IF bAConeOnMatrixConv AND bAutoModeOn AND bErrorReset AND NOT bIRowConeDetection  THEN
sMatrixConvStatus:='Continue Machine Operation '; bAConeOnMatrixConv:=FALSE;END_IF



(*===================== Auto Logic================*)


CASE step4 OF

	0:	IF( bARowStopperMotorRevStart ) AND bAutoModeOn THEN
		bAMove2_4Position:=FALSE;
		bAMove2_3Position:=FALSE;
		bRowStopperAt23Pos:=FALSE;
		bRowStopperAt24Pos:=FALSE;
		tRowStopperHomeDly(IN:=TRUE , PT:= t#1s , Q=> , ET=> );
		IF tRowStopperHomeDly.Q THEN   step4:=step4+1; END_IF
		END_IF

	1:	step4:=step4+1;


	2:	IF tRowStopperHomeDly.Q AND bAutoModeOn  AND NOT bAPauseSeq   THEN
		bQARowStopperMotorRevAuto:=TRUE;
		bARowStopperMotorRevStart:=FALSE;
		TON_2(IN:=FALSE);
		step4:=step4+1;
		END_IF

	3:	 step4:=step4+1;

	4:	IF bAutoModeOn AND bIRowStopperHome  THEN
		bQARowStopperMotorRevAuto:=FALSE;
		bAServoFwdStart:=TRUE;
		bAServoStartAuto:=TRUE;
		tRowStopperHomeDly(IN:=FALSE);
		step4:=step4+1;
		END_IF

	5:	 step4:=step4+1;

	6:	IF  bIGripperVerticalEnd THEN
		step4:=step4+1;
		END_IF

	7:	IF NOT bIGripperVerticalEnd   AND NOT bAPauseSeq   THEN
		step4:=step4+1;
		END_IF


	8:	 step4:=step4+1;

	9:	TON_2(IN:=TRUE , PT:=T#3S , Q=> , ET=> );
		IF TON_2.Q  THEN bAServoUpDone:=TRUE; step4:=step4+1; END_IF

	10:	 step4:=step4+1;


	11:	IF  bAutoModeOn AND  bAServoUpDone  AND b2_4SetHmiSelected THEN
		step4:=12;
		ELSIF  bAutoModeOn AND  bAServoUpDone AND b2_3SetHmiSelected THEN
		step4:=14;
		END_IF


	12:	 step4:=step4+1;

	13:	 bAMove2_4Position:=TRUE;
		step4:=16;

	14:	 step4:=step4+1;

	15:	bAMove2_3Position:=TRUE;
		step4:=step4+1;

	16:	 step4:=step4+1;

	17:	bAServoUpDone:=FALSE;
		step4:=0;

END_CASE

(*

R_TRIG_1(CLK:=b2_3SetHmiSelected , Q=> );


IF R_TRIG_1.Q AND NOT bIRowStopper2 THEN
b2_3FirstMoveStart:=TRUE;

END_IF

*)
(*
R_TRIG_2(CLK:=b2_4SetHmiSelected , Q=> );


IF R_TRIG_2.Q AND NOT bIRowStopper3 THEN
b2_4FirstMoveStart:=TRUE;

END_IF*)



(*============= Row Stopper Go to Home Logic While Servo Reset==========================*)


CASE Step5 OF
	0:	IF bRowStopperGoHome THEN bRowStopperGoRst:=TRUE; step5:=1; END_IF

	1:	IF bIRowStopperHome THEN  bRowStopperGoHome:=FALSE; bRowStopperGoRst:=FALSE; Step5:=0; END_IF

END_CASE


IF NOT bIEmergencySwitch OR bStopHmi   OR bServoOff OR bIMcStop  THEN
TON1temp4(IN:=FALSE);
RevStartT(IN:=FALSE);
bA2_4MoveEnable:=FALSE;
bA2_4RowMoveStarted:=FALSE;
bRowStopperAt24Pos:=FALSE;
bA2_3MoveEnable:=FALSE;
b23CheckDly(IN:=FALSE);
bA2_3MoveStarted:=FALSE;
TON_Mx(IN:=FALSE);
bRowStopperAt23Pos:=FALSE;
bRowStopperIntOver:=FALSE;
bAConeOnMatrixConv1:=FALSE;
bAConeOnMatrixConv2:=FALSE;
bAConeOnMatrixConv:=FALSE;
tRowStopperHomeDly(IN:=FALSE);
TON_2(IN:=FALSE);
bAServoFwdStart:=FALSE;
bAServoUpDone:=FALSE;
bAMove2_4Position:=FALSE;
bAMove2_3Position:=FALSE;

bQARowStopperMotorFwd1:=FALSE;
bQARowStopperMotorFwd2:=FALSE;
bQARowStopperMotorFwd3:=FALSE;
bQARowStopperMotorRev1:=FALSE;
bQARowStopperMotorRev2:=FALSE;
bQARowStopperMotorRev3:=FALSE;
bQARowStopperMotorRevAuto:=FALSE;
bRowStopperGoRst:=FALSE;
step2:=0;
step1:=0;
step3:=0;
step4:=0;

END_IF
END_PROGRAM

(* POU Auto/ColumStopperMotor, ST *)
PROGRAM ColumStopperMotor
VAR
	bQAColumnStopperMotorFwd1: BOOL;
	bQAColumnStopperMotorRev1: BOOL;
	step1: INT;

	test: BOOL;

	step2: INT;
	ColumnStopperInHome: BOOL;
	bA4_4MoveStarted: BOOL;
	bQAColumnStopperMotorFw21: BOOL;
	bQAColumnStopperMotorFwd2: BOOL;
	bQAColumnStopperMotorRev2: BOOL;
	bQAColumnStopperMotorFw2: BOOL;
	test1: BOOL;
	step3: INT;
	test2: BOOL;
	bA2_3MoveStarted: BOOL;
	bQAColumnStopperMotorRev3: BOOL;
	bQAColumnStopperMotorFwd3: BOOL;
	RevOffDly: TON;
	bA2_4MoveStarted: BOOL;
	Timer1: TON;
	Timer2: TON;
	bStopHmitemp: BOOL;
	bProgramChange: BOOL;
	bColumnStopMove2_3: BOOL;
	bColumnStopMove2_4: BOOL;
	b2_3SetHmiSelectedtemp: BOOL;
	b2_4SetHmiSelectedtemp: BOOL;
	b2_4SetHmiSelectedtemp1: BOOL;
	Mybit1: BOOL;
END_VAR
bQAColumnStopperMotorForward:= ( bQAColumnStopperMotorFwd1 OR bQAColumnStopperMotorFwd2 OR bQAColumnStopperMotorFwd3  ) ;
bQAColumnStopperMotorReverse:= ( bQAColumnStopperMotorRev1 ) ;

								(*=========== Column Stopper Motor Home Position Logic===============*)

CASE step2 OF

	0:	IF  bInitializeHmi AND bMCStartInAuto  AND NOT bIColumnStopperHome  AND NOT bAinterlockinit   THEN
		bQAColumnStopperMotorFwd1:=TRUE;
		(*	Timer1(IN:=TRUE  , PT:=t#1s , Q=> , ET=> );   *) step2:=step2+1;
		ELSIF  bInitializeHmi AND  bIColumnStopperHome    THEN   step2:=4;
		END_IF

	1:	bQAColumnStopperMotorFwd1:=FALSE;
		Timer2(IN:=TRUE , PT:= t#0.5s, Q=> , ET=> );
		IF Timer2.Q THEN step2 :=step2+1; END_IF

	2:	IF NOT bAPauseSeq  THEN  bQAColumnStopperMotorRev1:=TRUE; step2:=step2+1; END_IF

	3:	IF bIColumnStopperHome THEN bQAColumnStopperMotorRev1:=FALSE; step2:=step2+1; END_IF

	4:	IF b2_3SetHmiSelected THEN bColumnStopMove2_3:=TRUE; step2:=0;
		ELSIF b2_4SetHmiSelected THEN bColumnStopMove2_4:=TRUE; step2:=0;
		END_IF

END_CASE

										(*=========== Column Stopper Motor 2_3 Position Logic===============*)

CASE step1 OF

	0:	IF  b2_3SetHmiSelected AND bColumnStopMove2_3 AND NOT bIColumnStopper3  AND  bIColumnStopperHome  THEN
		 bQAColumnStopperMotorFwd2:=TRUE; step1:=step1+1;
		END_IF

	1:	IF bIColumnStopper3 THEN
	         bColumnStopMove2_3:=FALSE;
                  bQAColumnStopperMotorFwd2:=FALSE; step1:=step1+1;
		END_IF

	2:	 step1:=0;

END_CASE

										(*=========== Column Stopper Motor 2_4 Position Logic===============*)

CASE step3 OF

	0:	IF b2_4SetHmiSelected AND  bColumnStopMove2_4 AND NOT bIColumnStopper2  AND    bIColumnStopperHome   THEN
		bQAColumnStopperMotorFwd3:=TRUE; step3:=step3+1;
		END_IF


	1: 	IF bIColumnStopper2 THEN
		bColumnStopMove2_4:=FALSE;
		bQAColumnStopperMotorFwd3:=FALSE; step3:=step3+1;
		END_IF


	2:	step3:=0;

END_CASE
END_PROGRAM

(* POU StartUp/GripperUnitRst, ST *)
PROGRAM GripperUnitRst
VAR
	step: INT;
	bILengthTightPistonEnd: BOOL;
	bIBredthTightPistonEnd: BOOL;
	bEmptyCortonConveyoPiatonHome: BOOL;
	bHorPistonAtReadyPos: BOOL;
	bHorPistonAtHomePos: BOOL;
	bHorPistonAtMiddlePos: BOOL;
	bGripperAtHomePos: BOOL;
	bGripperAtEndPos: BOOL;
	bGripperAtMiddlePos: BOOL;
	bSepVerticalAtHomePos: BOOL;
	bSepVerticalAtEndPos: BOOL;
	bSepVerticalAtMiddlePos: BOOL;
	bLenghtTightPistonHomeNok: BOOL;
	bBreathtightPistonHomeNok: BOOL;
	bApplicatorHomeNok: BOOL;
	bReleaseApplicator: BOOL;
	step2: INT;
	Timer1: TON;
	Timer2: TON;
	Timer3: TON;
	Timer4: TON;
	ReadyToRelease: BOOL;
	Timer5: TON;
	bAResetHmitemp: BOOL;
	Timer6: TON;
	Timer7: TON;
	Timer8: TON;
	Timer9: TON;
	test: BOOL;
	BTEST1: BOOL;
	Timer10: TON;
	Timer20: TON;
	check1: BOOL;
	R_TRIG_50: R_TRIG;
END_VAR
VAR_INPUT
END_VAR
IF bInitializeHmi AND bAutoModeOn AND bMCStartInAuto THEN
step:=0;
END_IF



CASE step OF
	0:	 bHomingDone:=FALSE;
		step:=step+1;

	1:	step:=step+1;


	2:	IF  bAResetHmitemp OR bMatrixConvIntOver THEN step:=step+1;  END_IF

	3:	IF NOT bIGripperVerticalHome AND bIServoReady THEN
		bServoStopHmi:=FALSE;
		bServoPwrOff:=FALSE;
		  bRServoHome:=TRUE; step:=step+1;
		ELSIF bIGripperVerticalHome AND bIServoReady  THEN
		step:=step+3;
		END_IF

	4:	IF bHomingDone THEN
		bMatrixConvIntOver:=FALSE;
		 step:=step+1; END_IF

	5:	IF bQALengthTightPistonValve AND bQABreadthTightPistonValve THEN
		bHomingDone:=FALSE;
		step:=step+1;
		ELSIF bQALengthTightPistonValve AND NOT bQABreadthTightPistonValve THEN
		bQABreadthTightPistonValve:=FALSE;
		bQALengthTightPistonValve:=FALSE;
		bQMBreadthTightPistonValve:=FALSE;
		bQMLengthTightPistonValve:=FALSE;

		bHomingDone:=FALSE;

		END_IF
		IF bILengthTightPistonHome THEN
		bQAConeEjectionPistonValve:=FALSE;
		bQMConeEjectionPistonValve:=FALSE;
		IF bIConeEjectionPistonHome THEN
		step:=step+1;
		END_IF
		END_IF
	6:	bMatrixConvIntOver:=FALSE;
		IF bISeparatorHorizontalPistonEnd AND NOT  bISeparatorHorizontalPistonHome THEN
		bHorPistonAtReadyPos:=TRUE; bHorPistonAtHomePos:=FALSE; bHorPistonAtMiddlePos:=FALSE;
		step:=step+1;
		ELSIF NOT bISeparatorHorizontalPistonEnd  AND  bISeparatorHorizontalPistonHome THEN
		bHorPistonAtHomePos:=TRUE; bHorPistonAtReadyPos:=FALSE; bHorPistonAtMiddlePos:=FALSE;
		step:=step+1;
		ELSIF NOT bISeparatorHorizontalPistonEnd  AND  NOT bISeparatorHorizontalPistonHome THEN
		bHorPistonAtMiddlePos:=TRUE; bHorPistonAtHomePos:=FALSE; bHorPistonAtReadyPos:=FALSE;
		step:=step+1;
		END_IF

	7:	IF bHorPistonAtReadyPos THEN step:=8;
		ELSIF bHorPistonAtHomePos THEN step:=25;
		ELSIF bHorPistonAtMiddlePos THEN  step:=25; END_IF

	8:	(* iControlWord1:=0;*)
		step:=step+1;

	9:	(* iControlWord1:=6;*)
		step:=Step+1;
(*========Waiting for row stopper to home==========*)

	10:	IF bIRowStopperHome THEN step:=Step+1;
		ELSIF NOT bIRowStopperHome THEN bRowStopperGoHome:=TRUE;  step:=Step+1;  END_IF


	11:	IF  bIRowStopperHome THEN
		bHomingDone:=FALSE;
		bARampDisableAuto:=FALSE;
		bARampDisableAuto2:=FALSE;
		bARampDisableAuto3:=FALSE;
		bARampDisableAuto4:=FALSE;
		bARampDisableRst:= FALSE;
		bAGoCounterAuto:=FALSE;
		bAGoCounterAuto2:=FALSE;
		bAGoCounterAuto3:= FALSE;
		bAGoCounterAuto4:=FALSE;
		bAGoCounterRst :=FALSE;
		bServoVarEnable:=TRUE;

		step:=Step+1;
		END_IF

	12:	bARampDisableAuto3:=TRUE;
		bServoStopHmi:=FALSE;
		bServoPwrOff:=FALSE;
		bAGoCounterAuto3:=FALSE;
		 step:=Step+1;

	13:	iATargetCounteValAuto:=29000;
		step:=Step+1;

	14:	iASetFequencyAuto:=(*iAServoVelocityHmi*)1300;
		 step:=Step+1;


	15:	bAGoCounterAuto3:=TRUE;
		step:=Step+1;

	16:	Timer2(IN:=TRUE , PT:= t#100ms, Q=> , ET=> );
		IF Timer2.Q THEN  step:=Step+1; END_IF

	17:	bARampDisableAuto3:=FALSE;
		step:=Step+1;

	18:	step:=Step+1;

	19:	IF  bIGripperVerticalEnd THEN step:=Step+1; END_IF


	20:	 bARampDisableAuto3:=TRUE;
		step:=Step+1;

	21:	(*IF statusWord.10 THEN step:=Step+1; END_IF*) step:=Step+1;

	22:	bQABreadthTightPistonValve:=FALSE;
		bQALengthTightPistonValve:=FALSE;
		bQMBreadthTightPistonValve:=FALSE;
		bQMLengthTightPistonValve:=FALSE;
		 step:=Step+1;

	23:
		IF(* bILengthTightPistonHome AND*) bIBreadthTightPistonHome AND bIGripperVerticalEnd   THEN
		Timer10(IN:= TRUE, PT:=t#2s , Q=> , ET=> );
		IF Timer10.Q THEN
		 step:=Step+1; END_IF
		END_IF

	24:	bServoVarEnable:=FALSE;
		bRServoHome:=TRUE;
		IF bHomingDone THEN bGripperUnitOver:=TRUE;  step:=0; END_IF

(*========Reseting all auto and manual output and enabling Rst outpus===================*)

	25:	IF bIGripperVerticalHome THEN
		bQASeparatorHorizontalPistonValveFWD:=FALSE;
		bQASeparatorHorizontalPistonValveREV:=FALSE;
		bQMSeparatorHorizontalPistonValveRev:=FALSE;
		bQMSeparatorHorizontalPistonValveFwd:=FALSE;
		bHomingDone:=FALSE;
		step:=step+1;
		END_IF

	26:	bQRSeparatorHorizontalPistonValveREV:=TRUE;
		step:=step+1;

	27:	IF bISeparatorHorizontalPistonEnd THEN
		bReleaseApplicator:=TRUE;
		bQRSeparatorHorizontalPistonValveREV:=FALSE; step:=step+1; END_IF


	28:	IF ReadyToRelease THEN	step:=step+1; 	END_IF

	29:	Timer5(IN:=TRUE , PT:=t#1s , Q=> , ET=> );
		IF Timer5.Q THEN ReadyToRelease:=FALSE; step:=step+1; 	END_IF

	30:	bQMBreadthTightPistonValve:=FALSE;
		bQMLengthTightPistonValve:=FALSE;
		bQABreadthTightPistonValve:=FALSE;
		bQALengthTightPistonValve:=FALSE;
		step:=step+1;

	31:	IF bIBreadthTightPistonHome(* AND bILengthTightPistonHome*) THEN
		bRServoHome1:=TRUE;
		IF bHomingDone THEN
		iASetFequencyAuto:=0;
		iASetFequencyRst:=0;
		bGripperUnitOver:=TRUE;  step:=0;bServoEnableAuto:=FALSE; END_IF
		END_IF


END_CASE




CASE step2 OF

	0:	IF bReleaseApplicator  THEN
		Timer6(IN:=FALSE);
		Timer7(IN:=FALSE);
		step2:=step2+1;
		END_IF

	1:	IF bIRowStopperHome THEN step2:=step2+1;
		ELSIF NOT bIRowStopperHome THEN  bRowStopperGoHome1:=TRUE;  step:=Step+1;  END_IF


	2: 	IF bIRowStopperHome  THEN
		bReleaseApplicator:=FALSE;
		Timer8(IN:=FALSE);
		step2:=step2+1;
		END_IF

	3:	Timer6(IN:=TRUE , PT:=T#100ms , Q=> , ET=> );
		IF Timer6.Q THEN
		step2:=step2+1;
		END_IF

	4:	IF NOT bIGripperVerticalEnd AND bIRowStopperHome THEN
		(*=========Changing the servo Mode to Velocity mode=============*)
		Timer8(IN:=FALSE);
		Timer9(IN:=FALSE);
		bARampDisableAuto2:=FALSE;
		bARampDisableAuto3:=FALSE;
		bARampDisableAuto4:=FALSE;
		bServoVarEnabe2:=TRUE;

		step2:=step2+1;
		END_IF

	5:	bARampDisableAuto4:=TRUE;
		bAGoCounterAuto4:=FALSE;
		bServoStopHmi:=FALSE;
		bServoPwrOff:=FALSE;
		step2:=step2+1;

	6:	iATargetCounteValAuto:=29100;
		step2:=step2+1;

	7:	iASetFequencyAuto:=(*iAServoVelocityHmi*)1300;
		step2:=step2+1;

	8:	bAGoCounterAuto4:=TRUE;
		step2:=step2+1;

	9:	step2:=step2+1;


	10:	bARampDisableAuto4:=FALSE;
		step2:=step2+1;


	11:	 step2:=step2+1;


	12:	step2:=step2+1;


	13:	IF R_TRIG_50.Q THEN
		bARampDisableAuto4:=TRUE;
		bServoStopHmi:=TRUE;
		step2:=step2+1;
		END_IF

	14: 	Timer6(IN:=FALSE);
		Timer7(IN:=FALSE);
		Timer8(IN:=FALSE);
		Timer9(IN:=FALSE);
		Timer20(IN:=FALSE);
		step2:=step2+1;

	15:	ReadyToRelease:=TRUE;
		bServoVarEnabe2:=FALSE;

		step2:=0;




END_CASE


R_TRIG_50(CLK:=bIGripperVerticalEnd , Q=> );


IF NOT bIEmergencySwitch OR bStopHmi OR bIMcStop OR bServoOff  THEN

bRServoHome:=FALSE;
bHorPistonAtReadyPos:=FALSE;
bHorPistonAtHomePos:=FALSE;
bHorPistonAtMiddlePos:=FALSE;
bAModeWrite:=FALSE;
Timer1(IN:=FALSE);
Timer2(IN:=FALSE);
Timer3(IN:=FALSE);
Timer4(IN:=FALSE);
bRServoHome:=FALSE;
bQRSeparatorHorizontalPistonValveREV:=FALSE;
Timer5(IN:=FALSE);
bRServoHome1:=FALSE;
bReleaseApplicator:=FALSE;
bGripperUnitOver:=FALSE;
Timer6(IN:=FALSE);
Timer7(IN:=FALSE);
Timer8(IN:=FALSE);
Timer9(IN:=FALSE);
iControlWord1.4:= FALSE;
ReadyToRelease:=FALSE;
iControlWord1:=7;
step:=0;
step2:=0;
		(*bARampDisableAuto:=FALSE;
		bARampDisableAuto2:=FALSE;
		bARampDisableAuto3:=FALSE;
		bARampDisableAuto4:=FALSE;
		bARampDisableRst:= FALSE;
		bAGoCounterAuto:=FALSE;
		bAGoCounterAuto2:=FALSE;
		bAGoCounterAuto3:= FALSE;
		bAGoCounterAuto4:=FALSE;
		bAGoCounterRst :=FALSE;*)
END_IF
END_PROGRAM

(* POU Serial, ST *)
PROGRAM Serial
VAR
	bSendStr:BOOL;
	Timer: TON;
	TrigSend:R_TRIG;
	TransmitStr : SendString;
	SendBusy: BOOL;
	SendErrorID: ComError_t;

	ReceiveStr :ReceiveString;
	ReStr: STRING;
	LastReceivedString: STRING;
	StringReceived: BOOL;
	ReceiveBusy: BOOL;
	ReceiveError: BOOL;
	ReceiveErrorID: ComError_t;
	ReceiveTimeout: BOOL;
	ReceiveCounter: UDINT;

	(* Serial communication with the COM port device *)
	COMportControl: SerialLineControl;
	COMportControlError: BOOL;
	COMportControlErrorID: ComError_t;


	Decimaldata: BYTE;
	Stringdata: STRING;
	RxBufferStringdata: STRING(300);
         TxBufferStringdata: STRING(300);
	RxBufferArrdata: ARRAY [0..80] OF BYTE;
	TxBufferArrdata: ARRAY [0..80] OF BYTE :=(*16#0F, 16#FA, 16#03, 16#00, 16#0D, 16#00, 16#10, 16#20, 16#01, 16#05, 16#58, 16#DF, 16#98, 16#00, 16#00, 16#02, 16#04, 16#E0, 16#B4, 16#F0;*)
16#0F, 16#FA, 16#03, 16#00, 16#02, 16#00, 16#38, 16#24, 16#F0; (*16#00, 16#00, 16#00, 16#00;, 16#10, 16#20, 16#05, 16#02, 16#AF, 16#F6, 16#98, 16#00, 16#00, 16#02, 16#04, 16#E0, 16#84, 16#F0;*)
	i: INT;
	ReceiveData_1: ReceiveData;

	SReceivedataFormat: ARRAY [0..300] OF BYTE;
	SReceivedatStringFt: STRING(300);
	sSendString_1: STRING(300);
	TransmitArrByteData: SendData;
(*==============port 2==========*)
	ReceiveData_2: ReceiveData;

	test: BOOL;
	SReceivedataFormat_2: ARRAY [0..300] OF BYTE;

	SReceivedatStringFt_2: STRING(300);
	COMportControl_2: SerialLineControl;
	COMportControlError_2: BOOL;
	COMportControlErrorID_2: ComError_t;
	SReceivedatStringFtTemp: STRING(300);
	SReceivedatStringFt_2Temp: STRING(300);


	ReceiveData_3: ReceiveData;
	SReceivedataFormat_3: ARRAY [0..300] OF BYTE;
	SReceivedatStringFt_3: STRING(300);
	SReceivedatStringFt_3Temp: STRING(300);
	COMportControl_3: SerialLineControl;
	COMportControlError_3: BOOL;
	COMportControlErrorID_3: ComError_t;
	SReceivedatStringFtTemp_1: STRING(300);
	Weight: REAL;
	SReceivedatStringFtTemp_11: STRING(300);
	Reset_Timer: TON;
	Reset_value: INT;
	Reset_01: BOOL;
END_VAR
(*
TrigSend(CLK:=bSendStr , Q=> );

Timer(IN:=TRUE, PT:=T#1s);


IF TrigSend.Q THEN
	TransmitArrByteData(
	pSendData:= ADR(TxBufferArrdata),
	Length:=100 ,
	TXbuffer:= TxBuffer1,
	Busy=> ,
	Error=> );

	Timer(IN:=FALSE);

END_IF;



MEMCPY(ADR(sSendString), ADR(TxBufferArrdata), 50);
*)
(*==============El6002 serial Communication Program for Laod Cell value read in Rs232 port 1 ==================*)


COMportControl(
	Mode:= SERIALLINEMODE_EL6_22B,
	pComIn:= ADR(COMin_COMport),
	pComOut:= ADR(COMout_COMport),
	SizeComIn:= SIZEOF(COMin_COMport),
	TxBuffer:= TxBuffer1,
	RxBuffer:= RxBuffer1,
	Error=> COMportControlError,
	ErrorID=> COMportControlErrorID );

(************************************
MAIN.string_Dec();

***)



(*
FOR i:=0 TO 300 DO
	RxBufferStringData[i]:= RxBuffer1.Buffer[i];
END_FOR*)

ReceiveData_1(
	pPrefix:= ,
	LenPrefix:= ,
	pSuffix:= ,
	LenSuffix:= ,
	pReceiveData:=  ADR(SReceivedataFormat),
	SizeReceiveData:= SIZEOF(SReceivedataFormat),(*100*)
	Timeout:=t#1s ,
	Reset:= ,
	RXbuffer:=RxBuffer1 ,
	DataReceived=> ,
	busy=> ,
	Error=> ,
	RxTimeout=> ,
	LenReceiveData=> );

MEMCPY(ADR(SReceivedatStringFt), ADR(SReceivedataFormat), 22);

SReceivedatStringFt:=MID(STR:=SReceivedatStringFt, LEN:=7, POS:=3);

 rRetUnitAWeight:=STRING_TO_REAL (SReceivedatStringFt);

 rRetUnitAWeight_display:= (SReceivedatStringFt);


(*==============El6002 serial Communication Program for Laod Cell value read in Rs232 port 2 ==================*)

COMportControl_2(
	Mode:= SERIALLINEMODE_EL6_22B,
	pComIn:= ADR(COMin_2_COMport_2),
	pComOut:= ADR(COMout_2_COMport_2),
	SizeComIn:= SIZEOF(COMin_2_COMport_2),
	TxBuffer:= TxBuffer2,
	RxBuffer:= RxBuffer2,
	Error=> COMportControlError_2,
	ErrorID=> COMportControlErrorID_2 );
(*

 CASE Reset_value OF

	0:	Reset_01:=FALSE; Reset_value:=Reset_value+1;

	1:	Reset_Timer( IN:= (NOT Reset_01) , PT:=T#0.2S , Q=> , ET=> );
	      IF Reset_Timer.Q THEN Reset_value:=Reset_value+1; END_IF

	2:	Reset_Timer(IN:=FALSE); Reset_01:=TRUE;Reset_value:=0;

END_CASE*)



ReceiveData_2(
	pPrefix:= ,
	LenPrefix:= ,
	pSuffix:= ,
	LenSuffix:= ,
	pReceiveData:=  ADR(SReceivedataFormat_2),
	SizeReceiveData:=SIZEOF(SReceivedataFormat_2),(* 100,*)
	Timeout:=t#1s ,
	Reset:=Reset_01 ,
	RXbuffer:=RxBuffer2 ,
	DataReceived=> ,
	busy=> ,
	Error=> ,
	RxTimeout=> ,
	LenReceiveData=> );

MEMCPY(ADR(SReceivedatStringFtTemp), ADR(SReceivedataFormat_2), 22);

rRetUnitBWeight_2:=(*STRING_TO_REAL *)(SReceivedatStringFtTemp);

SReceivedatStringFtTemp:=MID(STR:=SReceivedatStringFtTemp, LEN:=7, POS:=3);


 rRetUnitBWeight:=STRING_TO_REAL (SReceivedatStringFtTemp);

 rRetUnitBWeight_Display:= (SReceivedatStringFtTemp);

(*MEMCPY(ADR(Weight), ADR(SReceivedatStringFt_2Temp), SIZEOF(SReceivedatStringFt_2Temp));*)


(*==============El6002 serial Communication Program for Laod Cell value read in Rs232 port 2 (  GROSS WEIGHT    )  ==================*)

COMportControl_3(
	Mode:= SERIALLINEMODE_EL6_22B,
	pComIn:= ADR(COMin_3_COMport_3),
	pComOut:= ADR(COMout_3_COMport_3),
	SizeComIn:= SIZEOF(COMin_3_COMport_3),
	TxBuffer:= TxBuffer3,
	RxBuffer:= RxBuffer3,
	Error=> COMportControlError_3,
	ErrorID=> COMportControlErrorID_3 );






ReceiveData_3(
	pPrefix:= ,
	LenPrefix:= ,
	pSuffix:= ,
	LenSuffix:= ,
	pReceiveData:=  ADR(SReceivedataFormat_3),
	SizeReceiveData:= SIZEOF(SReceivedataFormat_3),(* 100,*)
	Timeout:=t#1s ,
	Reset:= ,
	RXbuffer:=RxBuffer3 ,
	DataReceived=> ,
	busy=> ,
	Error=> ,
	RxTimeout=> ,
	LenReceiveData=> );

MEMCPY(ADR(SReceivedatStringFt_3), ADR(SReceivedataFormat_3), 22);

SReceivedatStringFt_3Temp:=MID(STR:=SReceivedatStringFt_3, LEN:=7, POS:=3);


 rGrossWeight:=STRING_TO_REAL (SReceivedatStringFt_3Temp);

 rGrossWeight_display:= (SReceivedatStringFt_3Temp);
END_PROGRAM

(* POU Auto/Gripper/Servo_Manual, ST *)
PROGRAM Servo_Manual
VAR
	step: INT;
	bAReset: BOOL;


	check: BOOL;
	Timer1: TON;
	btest: BOOL;
END_VAR
IF bManualModeOn THEN

bARampDisable:= (  bARampDisable_Man   );

bAGoCounter:= ( bAGoCounter_Man );

iASetFequency:=500;


bARampDisableAuto:=FALSE;
 bARampDisableAuto2:=FALSE;
 bARampDisableAuto3:=FALSE;
 bARampDisableAuto4:=FALSE;
bAGoCounterAuto:=FALSE;
 bAGoCounterAuto2:=FALSE;
 bAGoCounterAuto3:=FALSE;
 bAGoCounterAuto4:=FALSE;
bServoEnableAuto:=TRUE;
bServoStopHmi:=FALSE;
 bServoPwrOff:=FALSE;
 END_IF


IF NOT bJogPositiveHmi THEN
IF bManualModeOn AND ( bJogNegativeHmi OR bServoHomeHmi )AND NOT bJogPositiveHmi THEN
 bARampDisable_Man_1:=FALSE; bARampDisable_Man:=FALSE; bAGoCounter_Man:=TRUE; ELSE bARampDisable_Man_1:=TRUE; END_IF END_IF

IF NOT bJogNegativeHmi THEN
IF bManualModeOn AND  bJogPositiveHmi  AND NOT bJogNegativeHmi  AND NOT bIGripperVerticalEnd  THEN
bARampDisable_Man:=FALSE; bAGoCounter_Man:=FALSE; ELSE bARampDisable_Man:=TRUE; END_IF END_IF


IF bManualModeOn AND  bIGripperVerticalHome  THEN  bJogNegativeHmi:=FALSE; END_IF
END_PROGRAM

(* POU Auto/Gripper/Servo_Auto_1, ST *)
PROGRAM Servo_Auto_1
VAR
	step: INT;


	iASetFequencyFlag: UINT;

	bAServoDownDone1: BOOL;

	iAServoRevVelocityHmi: UINT := 6000;
	bAServoFwdStart1: BOOL;
	test: BOOL;


	step2: INT;
	test2: BOOL;
	test3: BOOL;
	iASetCounteVal2: UINT;
	bASetCounter2: BOOL;
	Count: INT;
	iTargetCounter: UINT;
	TON_1: TON;
	TON_14: TON;
	bAServoAutoStart_1: BOOL;
	R_TRIG_150: R_TRIG;
END_VAR
R_TRIG_150(CLK:=bIGripperVerticalEnd , Q=> );

IF bAutoModeOn AND CountServo = 0 THEN
iDropPosHmi:=iDropPos1Hmi;

ELSIF bAutoModeOn AND  CountServo=1 THEN
iDropPosHmi:=iDropPos2Hmi;
ELSIF bAutoModeOn AND  CountServo = 2 THEN
iDropPosHmi:=iDropPos3Hmi;
END_IF


IF bAServoHoming AND NOT bManualModeOn  THEN

bARampDisable:= (  bARampDisableRst  );

bAGoCounter:= ( bAGoCounterRst );

iASetCounteVal:= ( iASetCounteValRst );

bASetCounter:= (bASetCounterRst );

iATargetCounteVal:= (iATargetCounteValRst );

iASetFequency:=( iASetFequencyRst  );

END_IF



IF bAServoStartAuto OR bServoVarEnable OR bServoVarEnabe2 OR bAServoAutoStart_1 AND NOT bManualModeOn THEN

bARampDisable:=((bARampDisableAuto OR bARampDisableAuto2 OR bARampDisableAuto3 OR bARampDisableAuto4) AND NOT bManualModeOn) ;

bAGoCounter := ((bAGoCounterAuto OR bAGoCounterAuto2 OR bAGoCounterAuto3 OR bAGoCounterAuto4) AND NOT bManualModeOn);

iATargetCounteVal:= (iATargetCounteValAuto );

iASetFequency:=  iASetFequencyAuto  ;

bASetCounter:= ( bASetCounter2 );

iASetCounteVal:= ( iASetCounteVal2 );

END_IF




CASE step OF

	0:	IF bAServoFwdStart AND bAutoModeOn  AND bIGripperVerticalHome AND  bILengthTightPistonHome AND bIBreadthTightPistonHome
		AND bISeparatorHorizontalPistonEnd AND  bIRowStopperHome AND NOT  bIRowStopper2 AND NOT  bIRowStopper3    THEN
		bAServoHoming:=FALSE;
		bHomingDone:=FALSE;
		bARampDisableAuto2:=FALSE;
		bARampDisableRst:=FALSE;
		bAServoAutoStart_1:=TRUE;
		step:=Step+1;
		END_IF

	1: 	bARampDisableAuto:=TRUE;
		bAGoCounterAuto:=FALSE;
		step:=Step+1;

	2:	iATargetCounteValAuto:=(*rTargetPosFinal*)29000;
		step:=Step+1;

	3:	iASetFequencyAuto:=(*iAServoVelocityHmi*)rPickVeloFinal(*4000*);
		step:=Step+1;

	4:	bAGoCounterAuto:=TRUE;
		step:=Step+1;

	5:	bARampDisableAuto:=FALSE;
		bAServoFwdStart:=FALSE;
		TON_1(IN:=FALSE);
		step:=Step+1;


	6:	IF bIGripperVerticalEnd AND  NOT bAPauseSeq  THEN
		step:=Step+1;
		(*ELSIF NOT bIGripperVerticalEnd AND iATargetCounteValAuto = (*iActCounter*)iACounterVal THEN
		step:=1;*)
		END_IF

	7:	bARampDisableAuto:=TRUE;
		bAGoCounterAuto:=FALSE;
		bAServoDownDone:=TRUE;
		step:=Step+1;

	8:	IF bAConePickDone  AND  NOT bAPauseSeq  THEN
		step:=Step+1;
		END_IF

	9:	TON_1(IN:=TRUE , PT:= T#1s, Q=> , ET=> );(* bASrevoAutoHome:=TRUE; *)                        (* Speed up*)
		IF TON_1.Q THEN Step:=Step+1; END_IF


	10:	iATargetCounteValAuto:=0;
		step:=Step+1;

	11:	iASetFequencyAuto:=(*iAServoRevVelocityHmi*)5000;
		bAConePickDone:=FALSE;
		step:=Step+1;

	12:	bAGoCounterAuto:=TRUE;
		step:=Step+1;

	13:	bARampDisableAuto:=FALSE;
		TON_1(IN:=FALSE);
		step:=Step+1;

	14:	IF bIGripperVerticalHome AND  NOT bAPauseSeq THEN

		Step:=Step+1;
		ELSIF NOT bIGripperVerticalHome AND iACounterVal = 0 THEN

		 Step:=1;
		END_IF


	15:	bARampDisableAuto:=TRUE;
		bAGoCounterAuto:=FALSE;
		bServoReachedUp:=TRUE;

		Step:=0;

END_CASE






CASE step2 OF

	0:	IF bAServoFwdStart2 AND bAutoModeOn AND bIGripperVerticalHome  AND bISeparatorHorizontalPistonHome THEN
		bARampDisableAuto:=FALSE;
		bARampDisableRst:=FALSE;
		bAServoHoming:=FALSE;
		step2:=Step2+1;
		END_IF

	1: 	bARampDisableAuto2:=TRUE;
		bAGoCounterAuto2:=FALSE;
		step2:=Step2+1;

	2:	iATargetCounteValAuto:=REAL_TO_UINT(rDropPosFinal);
		step2:=Step2+1;

	3:	iASetFequencyAuto:= REAL_TO_UINT(rDropVeloFinal)(*iAServoVelocityHmi    1500*);
		step2:=Step2+1;

	4:	bAGoCounterAuto2:=TRUE;
		step2:=Step2+1;

	5:	bARampDisableAuto2:=FALSE;
		bAServoFwdStart2:=FALSE;
		step2:=Step2+1;


	6:	IF CountServo=0 AND  iACounterVal >=23600 THEN
		step2:=Step2+1;
		ELSIF CountServo=1 AND   iACounterVal >=17300 THEN
		step2:=Step2+1;
		ELSIF CountServo=2 AND   iACounterVal >=12245 THEN
		step2:=Step2+1;
		END_IF

	7:	bARampDisableAuto2:=TRUE;
		bAGoCounterAuto2:=FALSE;
		bAServoDown1Done:=TRUE;
		step2:=Step2+1;

	8:	IF  bAServoUpAuto  THEN
		step2:=Step2+1;
		END_IF

	9:	(* bASrevoAutoHome:=TRUE; *)TON_14(IN:=TRUE , PT:= t#1s, Q=> , ET=> );
		IF TON_14.Q THEN  step2:=Step2+1; END_IF

	10:	iATargetCounteValAuto:=0;
		step2:=Step2+1;

	11:	iASetFequencyAuto:=(*iAServoRevVelocityHmi*)5000;
		bAServoUpAuto:=FALSE;
		step2:=Step2+1;

	12:	bAGoCounterAuto2:=TRUE;
		step2:=Step2+1;

	13:	IF bAutoModeOn THEN
		bARampDisableAuto2:=FALSE;
		step2:=Step2+1;
		END_IF
	14:	IF bIGripperVerticalHome THEN
		Step2:=Step2+1;
		END_IF


	15:	bARampDisableAuto2:=TRUE;
		bAGoCounterAuto2:=FALSE;
		TON_14(IN:=FALSE);
		Step2:=Step2+1;

	16:	IF iACounterVal =0  THEN step2:=3;
		ELSIF iACounterVal <> 0   THEN Step2:=Step2+1; END_IF

	17:	iASetCounteVal2:=0;
		step2:=Step2+1;

	18:	bASetCounter2:=TRUE;
		IF  iActCounter = 0 THEN step2:=Step2+1; END_IF

	19:	bASetCounter2:=FALSE;
		bAPlaceOver:=TRUE;

		step2:=Step2+1;

	20:	CountServo:=CountServo+1;
		step2:=Step2+1;

	21: IF CountServo=3 THEN
		iACountServoToSepUnit:= CountServo;
		CountServo:=0;
		step2:=Step2+1;
		ELSIF CountServo<3 THEN
		step2:=Step2+1;
		END_IF

	22:	step2:=0;		bAServoAutoStart_1:=FALSE;



END_CASE

(*
IF  bIEmergencySwitch THEN
bQServoEnable:=TRUE;
ELSE
bQServoEnable:=FALSE;
END_IF

*)



IF bAutoModeOn AND Count = 0 THEN
iTargetCounter:=29000;
ELSIF bAutoModeOn AND  Count=1 THEN
iTargetCounter:=15000;
ELSIF bAutoModeOn AND  Count = 2 THEN
iTargetCounter:=10000;
END_IF


IF  NOT bIEmergencySwitch OR bStopHmi OR bServoOff  OR bIMcStop THEN
bServoStopHmi:=TRUE;
bARampDisableAuto :=FALSE;
bARampDisableAuto2 :=FALSE;
bARampDisableAuto3 :=FALSE;
 bARampDisableAuto4:=FALSE ;

bAGoCounterAuto :=FALSE;
bAGoCounterAuto2 :=FALSE;
 bAGoCounterAuto3 :=FALSE;
bAGoCounterAuto4:=FALSE;;

 bARampDisableRst:=FALSE;
bAGoCounterRst:=FALSE;

bASetCounterRst:=FALSE;
step:=0;
step2:=0;
Count:=0;
iASetFequencyAuto:=0;
iASetFequency:=0;
bAServoAutoStart_1:=FALSE;
bServoVarEnable:=FALSE;
bServoVarEnabe2:=FALSE;
END_IF
END_PROGRAM

(* POU Auto/Gripper/PickAndPlaceUnit, ST *)
PROGRAM PickAndPlaceUnit
VAR
	step: INT;
	tL_BPistonCloseDly: TON;
	bIGripperVerticalHomeTemp: BOOL;
	test: BOOL;
	bAServoDownDone1: BOOL;
	TON_1: TON;
	bIConeEjectionPistonEndtemp: BOOL;
	bIConeEjectionPistonHomeTemp: BOOL;
	Timer1: TON;
	Timer2: TON;
	SepHoriCylHomeRsErrChk: RS_Error;
	SepHoriCylHomeRsErr: BOOL;
	SepHoriCylEndRsErrChk: RS_Error;
	SepHoriCylEndRsErr: BOOL;
END_VAR
	IF NOT  bIEmergencySwitch OR   bStopHmi OR bServoOff OR bIMcStop THEN
	tL_BPistonCloseDly(IN:=FALSE);
	Timer2(IN:=FALSE);
	step:=0;
	bQASeparatorHorizontalPistonValveREV:=FALSE;
	(*bQALengthTightPistonValve:=FALSE;
	bQABreadthTightPistonValve:=FALSE;
	 bAConePickDone:=FALSE;*)
	bAServoDownDone:=FALSE;
	Timer1(IN:=FALSE);
	bQASeparatorHorizontalPistonValveFWD:=FALSE;
	TON_1(IN:=FALSE);
	bAServoFwdStart2:=FALSE;
	(*bQAConeEjectionPistonValve:=FALSE;*)
	bAServoDown1Done:=FALSE;
	bAServoUpAuto:=FALSE;
	bServoReachedUp:=FALSE;
	bAPlaceOver:=FALSE;
END_IF


CASE step OF

	0:	tL_BPistonCloseDly(IN:=FALSE);
		Timer2(IN:=FALSE);
		 step:=step+1;

	1:	 step:=step+1;

	2:	IF bAutoModeOn AND bAServoDownDone (*AND bILengthTightPistonHome*) AND bIBreadthTightPistonHome THEN
		tL_BPistonCloseDly(IN:=TRUE , PT:=T#0.2s , Q=> , ET=> );
		IF tL_BPistonCloseDly.Q THEN   step:=step+1;END_IF
		END_IF

	3:	 step:=step+1;

	4:	IF bAutoModeOn AND bAServoDownDone (*AND bILengthTightPistonHome*) AND bIGripperVerticalEnd   AND bIBreadthTightPistonHome
		AND  NOT bAPauseSeq  AND NOT bAL_BTightHomeSenRsError THEN
		bQASeparatorHorizontalPistonValveREV:=FALSE;
		bQALengthTightPistonValve:=TRUE;
		bQABreadthTightPistonValve:=TRUE;
		 step:=step+1;
		END_IF

	5:	Timer2(IN:=TRUE , PT:=t#2s , Q=> , ET=> );bAServoDownDone:=FALSE;
		IF Timer2.Q THEN  bAConePickDone:=TRUE; step:=step+1; END_IF

	6:	IF bAutoModeOn AND bIGripperVerticalHome AND bServoReachedUp AND bISeparatorHorizontalPistonEnd  AND bISeparatorVerticalPistonHome
		 AND (bACartonReady_23 OR bACartonReady_24) AND  NOT bAPauseSeq  AND NOT bIGripperVerticalEnd THEN
		bQASeparatorHorizontalPistonValveFWD:=TRUE;
		TON_1(IN:=FALSE);
		Timer2(IN:=FALSE);
		tL_BPistonCloseDly(IN:=FALSE);
		step:=step+1;
		END_IF

	7:	 step:=step+1;

	8:	IF  bAutoModeOn  AND bISeparatorHorizontalPistonHome  AND NOT bHmiColourChangeBit2_24 AND NOT bASepaHoriForwdEndRsError  AND NOT SeparatorAlertbit THEN

		(*bACartonReady_24:=FALSE;*)
		bServoReachedUp:=FALSE;
		TON_1(IN:=TRUE , PT:=t#0.3s  , Q=> , ET=> );
		IF TON_1.Q THEN step:=step+1; END_IF
		END_IF

	9:	 step:=step+1;

	10:	IF NOT bAPauseSeq THEN bAServoFwdStart2:=TRUE;
		 step:=step+1;
		END_IF

	11:	 step:=step+1;

	12:	IF  bAutoModeOn  AND bISeparatorHorizontalPistonHome  AND bAServoDown1Done  AND NOT bAPauseSeq THEN
		(*bQALengthTightPistonValve:=FALSE;*)
		bQABreadthTightPistonValve:=FALSE;
		step:=step+1;
		END_IF

	13:	 step:=step+1;

	14:	IF  bAutoModeOn AND bIConeEjectionPistonHome AND NOT bAPauseSeq  THEN
		bQAConeEjectionPistonValve:=TRUE;
		bAServoDown1Done:=FALSE;
		step:=step+1;
		END_IF

	15:	timer1(IN:=TRUE , PT:=T#0.5s , Q=> , ET=> );
		IF  timer1.Q   THEN step:=step+1; END_IF

	16:	IF  bAutoModeOn  THEN

		bAServoUpAuto:=TRUE;
		step:=step+1;
		END_IF

	17:	 step:=step+1;

	18:	IF bAutoModeOn AND  bIGripperVerticalHome (*AND statusWord.10  *)THEN
		(*bQABreadthTightPistonValve:=FALSE;*)
		bQALengthTightPistonValve:=FALSE;
		bQASeparatorHorizontalPistonValveFWD:=FALSE;
		step:=step+1;
		END_IF

	19:	 step:=step+1;

	20:	 IF bIBreadthTightPistonHome(* AND bILengthTightPistonHome*)  AND NOT bAPauseSeq  AND NOT bAL_BTightHomeSenRsError  THEN
		 bQAConeEjectionPistonValve:=FALSE;
		step:=step+1;
		END_IF

	21:	 step:=step+1;

	22:	IF bAPlaceOver AND bIGripperVerticalHome  AND bISeparatorVerticalPistonHome AND NOT bAPauseSeq  THEN
		bQASeparatorHorizontalPistonValveREV:=TRUE;
		step:=step+1;
		END_IF

	23:	step:=step+1;

	24:	IF bISeparatorHorizontalPistonEnd  AND NOT bASepaHoriRevValveRsError THEN
		bAServoStartAuto:=FALSE;
		bAPlaceOver:=FALSE;
		step:=0;
		END_IF

END_CASE
END_PROGRAM

(* POU FunctionBlocks/RS_Error, ST *)
FUNCTION_BLOCK RS_Error
VAR_INPUT
	bValveOutOn: BOOL;
	bReedSwithIn: BOOL;
	bErroReset: BOOL;
	sMsgIn: STRING;
	RS_ErrChkDly: TIME;
END_VAR
VAR_OUTPUT
	bRsError: BOOL;
	sMsgOut: STRING;
END_VAR
VAR
	FbStep: INT;
	Timer1: TON;
END_VAR
CASE FbStep OF


	0:	Timer1(IN:=FALSE); FbStep:=FbStep+1;

	1:	IF bValveOutOn THEN FbStep:=FbStep+1; END_IF

	2:	Timer1(IN:=TRUE , PT:=RS_ErrChkDly , Q=> , ET=> );
		IF Timer1.Q THEN FbStep:=FbStep+1;
		ELSIF NOT  Timer1.Q AND bReedSwithIn THEN  FbStep:=0; END_IF

	3:	IF bReedSwithIn THEN  FbStep:=FbStep+1;
		ELSIF NOT bReedSwithIn THEN FbStep:=FbStep+2; END_IF

	4:	IF  NOT bValveOutOn THEN sMsgOut:=sMsgIn;  FbStep:=0; END_IF

	5:	bRsError:=TRUE; FbStep:=FbStep+1;

	6:	IF   bReedSwithIn AND   bErroReset THEN bRsError:=FALSE; sMsgOut:='' ;  FbStep:=0;
		ELSIF   NOT bReedSwithIn AND   bRsError  AND  bErroReset THEN bRsError:=FALSE;   sMsgOut:='' ;   FbStep:=0;
		 END_IF

END_CASE
END_FUNCTION_BLOCK

(* POU Auto1/DataLog/DataLog_1, ST *)
PROGRAM DataLog_1
VAR
	stStation1_ProductionData: Production_Data;
	ST1_ProductionDataValues: STRING(3000);
	S1_iCyc_Count_DISP: INT;
	S1_iACT_HLD_TIMEDISP: INT;
	stActiveuserCredential: BOOL;
	nPressureMaxvalue: REAL;
	OperatorName: STRING;
	nMinimumTopTempLimit_ST1: INT;
	nMaximumTopTempLimit_ST1: INT;
	nTOPTempMaxvalue: UINT;
	nMinimumBTMTempLimit_ST1: INT;
	nBTMTempMaxvalue: UINT;
	nMaximumBTMTempLimit_ST1: INT;
	Set_HLDTIME: INT;
	S_1_iPressure: REAL;
	rS_PressureRange1: REAL;
	nMaxEnergy: REAL;
	nMaxPower: REAL;
	S_iSET_COUNT: INT;
	S1_iTotCyc_Count_DISP: INT;
	sJobStatus_ST1: STRING;
	sStation1_ProductionData_FileName: STRING(80) := 'Hard Disk\Reports\Test1\ProductionData.csv';
	Fb_LoagProductionData: DATA_LOG_Save;
	SaveData: BOOL;
	ST1_ProductionData: STRING(500);
	Fb_CreateFileFormat_1: Fb_CreateFileFormat;
	bEnableFileFormat: BOOL;
	wTodayTemp: STRING;
	sDateTemp: STRING;
	sOLDFileName_ST1: T_MaxString;
	Fb_FormatDrive_1: Fb_FormatDrive;
	bFileDelete: BOOL;
	Fb_CopyBackupAL_Server_LogOf_1: Fb_CopyFileToRemotePC;
	bool2: BOOL;
	bAstart: BOOL;
	TON_1: TON;
	TON_2: TON;
	CTU_1: CTU;
	R_TRIG_1: R_TRIG;
	R_TRIG_2: R_TRIG;
	bACreateNewFile: BOOL;
	ReportStep: INT;
	bANewDay: BOOL;
	Timer1: TON;
	Timer2: TON;
	R_TRIG1: R_TRIG;


	iUnitBNetWtTemp1: REAL;
	rRetUnitBWeightTemp1: REAL;
	StepTemp1: INT;
	rRetUnitBWeightTemp2: REAL;
	StepTemp2: INT;
	BCreateDir: BOOL;
	FB_CreateDir_1: FB_CreateDir;
	bANewDaytemp: BOOL;
	bit2: BOOL;
	hfile: UINT;
	FB_FileOpen_1: FB_FileOpen;
	test: BOOL;
	bit3: BOOL;
	FB_FileWrite_1: FB_FileWrite;
	bEnableFileFormattemp: BOOL;
	BDelete: BOOL;
	FB_FileDelete_1: FB_FileDelete;
	Timer3: TON;
	iCartoNoHmiTemp: DWORD;
	dateInint: WORD;
	E_OpenPath: E_OpenPath;
	FB_FileDelete_2: FB_FileDelete;
END_VAR
FileCreateTemp;

Fb_CreateFileFormat_1(
	sInputMessage:=ST1_ProductionData ,
	sFileName:='ProductionData' ,
	sDirectory:= '\\ACHME-PC\Reports\' (*  'Hard Disk\Reports\Indo\'  *) ,
	bEnable:=bEnableFileFormat ,
	wToday:=wTodayTemp ,
	sDate=> sDateTemp,
	bNewDateFound=> bANewDay,
	sOldFileName=>sOLDFileName_ST1 ,
	sFilePathFinal=> );

FB_FileDelete_2(
	sNetId:='169.254.147.163.1.1' ,
	sPathName:= sStation1_ProductionData_FileName ,
	ePath:=E_OpenPath ,
	bExecute:=bFileDelete ,
	tTimeout:=t#1s ,
	bBusy=> ,
	bError=> ,
	nErrId=> );


bLoadPgm;
IF (bloadRecipeHmi OR bSaveRecipeHmi) THEN
iCartoNoHmiTemp:=iCartoNoHmi;
ELSE
iCartoNoHmiTemp:=(ITotalSample +iCartoNoHmi);
END_IF

iCartonSample:=iCartoNoHmiTemp;

		stStation1_ProductionData.S_No						:=INT_TO_STRING( Pgm_NoHmi );
		stStation1_ProductionData.CartonNo					:=DWORD_TO_STRING(iCartoNoHmiTemp);
		stStation1_ProductionData.SDateF					:= (sDATEFinal);
		stStation1_ProductionData.sShift						:=(sShitToReport);
	(*	stStation1_ProductionData.ActualNetWt				:=REAL_TO_STRING(rRetUnitAWeight); *)
		stStation1_ProductionData.LotNo					:=(*DWORD_TO_STRING*)(iLotNoHmi);
		stStation1_ProductionData.sCount					:=(iCountHmi);
		stStation1_ProductionData.NetWt					:=REAL_TO_STRING(var_5);
		stStation1_ProductionData.StandardGrossWt			:=(var_7);
		stStation1_ProductionData.sTolerance				:=REAL_TO_STRING(NetToleranceHmi);
		stStation1_ProductionData.sEmpConeWt				:=REAL_TO_STRING(iWeightHmi);




		(*	######## LOG PRODUCTION DATA		#####	*)

ST1_ProductionDataValues:= CONCAT(stStation1_ProductionData.S_No,',');
ST1_ProductionDataValues:=	 CONCAT( ST1_ProductionDataValues,stStation1_ProductionData.CartonNo);
ST1_ProductionDataValues:= CONCAT( ST1_ProductionDataValues,',');
ST1_ProductionDataValues:=	 CONCAT( ST1_ProductionDataValues,stStation1_ProductionData.SDateF	);
ST1_ProductionDataValues:= CONCAT( ST1_ProductionDataValues,',');
ST1_ProductionDataValues:=	 CONCAT( ST1_ProductionDataValues,stStation1_ProductionData.sShift	);
ST1_ProductionDataValues:= CONCAT( ST1_ProductionDataValues,',');
(*ST1_ProductionDataValues:=	 CONCAT( ST1_ProductionDataValues,stStation1_ProductionData.ActualNetWt	);
ST1_ProductionDataValues:= CONCAT( ST1_ProductionDataValues,',');*)
ST1_ProductionDataValues:=	 CONCAT( ST1_ProductionDataValues,stStation1_ProductionData.LotNo);
ST1_ProductionDataValues:= CONCAT( ST1_ProductionDataValues,',');
ST1_ProductionDataValues:=	 CONCAT( ST1_ProductionDataValues,stStation1_ProductionData.sCount);
ST1_ProductionDataValues:= CONCAT( ST1_ProductionDataValues,',');
ST1_ProductionDataValues:=	 CONCAT( ST1_ProductionDataValues,stStation1_ProductionData. NetWt );
ST1_ProductionDataValues:= CONCAT( ST1_ProductionDataValues,',');
ST1_ProductionDataValues:=	 CONCAT( ST1_ProductionDataValues,stStation1_ProductionData.StandardGrossWt);
ST1_ProductionDataValues:= CONCAT( ST1_ProductionDataValues,',');
ST1_ProductionDataValues:=	 CONCAT( ST1_ProductionDataValues,stStation1_ProductionData.sEmpConeWt);
ST1_ProductionDataValues:= CONCAT( ST1_ProductionDataValues,'$0A');     (**)

(*==========Saving the Data to Report===========*)

sStation1_ProductionData_FileName:= Fb_CreateFileFormat_1.sOldFileName ; (*    'Hard Disk\Reports\Test1\ProductionData.csv' ;*)


Fb_LoagProductionData(
	bStartDataLog:= SaveData ,
	sDataLogFileName:=sStation1_ProductionData_FileName ,
	LogData:=ST1_ProductionDataValues ,
	bErrorDataLog=> );






(*=============== file copy from CX Controller to Remote PC & File Delete In CX Device======================*)


	Fb_CopyBackupAL_Server_LogOf_1(
		bMakeDirectory:= ,
		bCopyFile:=bool2,
		sDestDriveName:= '\\ACHME-PC\Reports\' ,
		sSourceDirectory:='\Hard Disk\Reports\Indo' ,
		 );

(*\\ramrajg-nb2\Ramaraj_public\   *)

  (*Hard Disk\Reports\  *)

Fb_FormatDrive_1(sDriveName:='\\ACHME-PC\Reports\' , bFormatDisk:=bFileDelete );


CASE ReportStep OF

	0:	 IF R_TRIG1.Q   THEN  FileCreateTemp:=TRUE; Timer3(IN:=FALSE); ReportStep:=1; END_IF

	1:	(*		##### Station 1 Production Data	#####	*)

		ST1_ProductionData:= CONCAT( 'Prg No',',');
		ST1_ProductionData:=	 CONCAT( ST1_ProductionData,'Carton No');
		ST1_ProductionData:= CONCAT( ST1_ProductionData,',');
		ST1_ProductionData:=	 CONCAT( ST1_ProductionData,'Date');
		ST1_ProductionData:= CONCAT( ST1_ProductionData,',');
		ST1_ProductionData:=	 CONCAT( ST1_ProductionData,'Shift');
		ST1_ProductionData:= CONCAT( ST1_ProductionData,',');
	(*	ST1_ProductionData:=	 CONCAT( ST1_ProductionData,'Unit');
		ST1_ProductionData:= CONCAT( ST1_ProductionData,',');*)
		ST1_ProductionData:=	 CONCAT( ST1_ProductionData,'Lot No');
		ST1_ProductionData:= CONCAT( ST1_ProductionData,',');
		ST1_ProductionData:=	 CONCAT( ST1_ProductionData,'Count');
		ST1_ProductionData:= CONCAT( ST1_ProductionData,',');
		ST1_ProductionData:=	 CONCAT( ST1_ProductionData,'Net Weight');
		ST1_ProductionData:= CONCAT( ST1_ProductionData,',');
		ST1_ProductionData:=	 CONCAT( ST1_ProductionData,'Gross Weight');
		ST1_ProductionData:= CONCAT( ST1_ProductionData,',');
		ST1_ProductionData:=	 CONCAT( ST1_ProductionData,'Tolerance');
		ST1_ProductionData:= CONCAT( ST1_ProductionData,',');
		ST1_ProductionData:=	 CONCAT( ST1_ProductionData,' Empty Cone Weight');
		ST1_ProductionData:= CONCAT( ST1_ProductionData,'$0A');

		ReportStep:=2;

	2:	Timer1(IN:=FALSE);
		bANewDay:=FALSE;
		ReportStep:=3;


	3:	bEnableFileFormat:=TRUE;
		Timer1(IN:=TRUE , PT:=T#100ms , Q=> , ET=> );
		IF Timer1.Q THEN bEnableFileFormat:=FALSE;  ReportStep:=4; END_IF


	4:	(*IF R_TRIG1.Q THEN  *)
		SaveData:=TRUE;
		Timer1(IN:=FALSE);
		ReportStep:=5;

	5:	Timer3(IN:=TRUE , PT:=T#20s , Q=> , ET=> );
		IF Timer3.Q THEN SaveData:=FALSE;bFileDelete:=TRUE;  ReportStep:=6; END_IF

	6:	 bFileDelete:=FALSE;Timer3(IN:=FALSE); FileCreateTemp:=FALSE; ReportStep:=0;

END_CASE



R_TRIG1(CLK:=(bACyclePass OR CyclePassTest)  , Q=> );


CASE StepTemp1 OF
	0:	IF bRetUnitBStart THEN rRetUnitBWeightTemp1:=rRetUnitBWeight; StepTemp1:=StepTemp1+1; END_IF

	1:	IF UnitBCompleteCheckCount.CV = 18 AND bAutoModeOn THEN rRetUnitBWeightTemp2:=rRetUnitBWeightTemp1;  StepTemp1:=0; END_IF
 END_CASE




CASE StepTemp2 OF
	0:	IF bRetUnitBStart THEN rRetUnitBWeightTemp1:=rRetUnitBWeight; StepTemp2:=StepTemp2+1; END_IF

	1:	IF c18_ConeCounter1.CV = 18 AND bAutoModeOn THEN rRetUnitBWeightTemp2:=rRetUnitBWeightTemp1; c18_ConeCounter1.RESET:=TRUE;  StepTemp2:=StepTemp2+1; END_IF

	2:	c18_ConeCounter1.RESET:=FALSE;  StepTemp2:=0;
 END_CASE
END_PROGRAM

(* POU FunctionBlocks/DATA_LOG_Save, ST *)
FUNCTION_BLOCK DATA_LOG_Save
VAR_INPUT
	bStartDataLog: BOOL;
	sDataLogFileName: STRING;
	LogData: STRING(1024);

END_VAR
VAR_OUTPUT

	bErrorDataLog: BOOL;
END_VAR
VAR

	R_TRIGStartDataLog: R_TRIG;
	nstep: INT;

	FB_OpenFile_Datalog: FB_FileOpen;
	nFB_OpenFile_Datalog_Errid: UDINT;

	FB_WriteFile_Datalog: FB_FileWrite;
	nFB_WriteFile_Datalog_ErrId: UDINT;

	FB_CloseFile_Datalog: FB_FileClose;
	nFB_CloseFile_Datalog_ErrId: UDINT;
	hDataLogSrcFile: UINT;

END_VAR
R_TRIGStartDataLog(CLK:=bStartDataLog , Q=> );
IF R_TRIGStartDataLog.Q THEN
		nstep :=1;
	END_IF

CASE nstep OF

	0:
		;
		FB_OpenFile_Datalog.bExecute:=FALSE;
		FB_WriteFile_Datalog.bExecute:=FALSE;
		FB_CloseFile_Datalog.bExecute:=FALSE;

	1:		(* do nothing *)
			nstep:=nstep+1;

	2:		(* ####	File Open ####*)

			FB_OpenFile_Datalog(  bExecute := FALSE  );
			FB_OpenFile_Datalog(	sNetId :='169.254.147.163.1.1' ,
			sPathName := sDataLogFileName,
			nMode := FOPEN_MODEAPPEND    ,
			ePath := PATH_GENERIC,
			tTimeout := T#2s,
			bExecute := TRUE );
			nstep := nstep+ 1;



	3:		FB_OpenFile_Datalog( bExecute := FALSE );
			IF ( NOT FB_OpenFile_Datalog.bBusy ) THEN
			IF ( FB_OpenFile_Datalog.bError ) THEN
			nFB_OpenFile_Datalog_Errid := FB_OpenFile_Datalog.nErrId;
			bErrorDataLog := TRUE;
			nstep := 50;
			ELSE
			hDataLogSrcFile := FB_OpenFile_Datalog.hFile;
			nstep := nstep + 1;
			END_IF
			END_IF

	4:		(*write data to destination file*)
			(*num:=num+1;*)
			FB_WriteFile_Datalog( bExecute := FALSE );
			FB_WriteFile_Datalog(	sNetId:='169.254.147.163.1.1',
			hFile:=FB_OpenFile_Datalog.hFile,
			pWriteBuff:= ADR(LogData),
			cbWriteLen:= LEN(LogData),		(*	i_len,	*)
			bExecute:=TRUE,
			tTimeout:=T#2s );
			nstep := nstep + 1;

	5:		FB_WriteFile_Datalog( bExecute := FALSE );
			IF ( NOT FB_WriteFile_Datalog.bBusy ) THEN
			IF ( FB_WriteFile_Datalog.bError ) THEN
			nFB_WriteFile_Datalog_ErrId := FB_WriteFile_Datalog.nErrId;
			bErrorDataLog := TRUE;
			nstep := 50;
			ELSE
			hDataLogSrcFile := FB_OpenFile_Datalog.hFile;
			nstep := nstep + 1;
			END_IF
			END_IF

	6:		(* close the destination file *)
			FB_CloseFile_Datalog( bExecute := FALSE );
			FB_CloseFile_Datalog( 	sNetId:='169.254.147.163.1.1' ,
			hFile:=FB_OpenFile_Datalog.hFile,
			bExecute:=TRUE,
			tTimeout:=T#2s );
			nstep := nstep + 1;

	7:		FB_CloseFile_Datalog( bExecute := FALSE );
			IF ( NOT FB_CloseFile_Datalog.bBusy ) THEN
			IF ( FB_CloseFile_Datalog.bError ) THEN
			nFB_CloseFile_Datalog_ErrId := FB_CloseFile_Datalog.nErrId;
			bErrorDataLog := TRUE;
			END_IF
			nstep := 0;
			END_IF

END_CASE
END_FUNCTION_BLOCK

(* POU FunctionBlocks/Fb_CreateFileFormat, LD *)
FUNCTION_BLOCK Fb_CreateFileFormat
VAR
	Fb_OpenFile: FB_FileOpen;
	Fb_WriteFile: FB_FileWrite;
	F_Trig1: F_TRIG;
	F_Trig2: F_TRIG;
	Fb_closeFile: FB_FileClose;
	F_Trig3: F_TRIG;


	SysteMtime: FB_LocalSystemTime;
	stSystemtimeAlrm: Timestruct;

	sFileName_Temp: T_MaxString;


	bCreateFileTrig: R_TRIG;
	bCreateFile: BOOL;
	Fb_SavePersistant: FB_WritePersistentData;
	TuneparaSave: BOOL;
END_VAR
VAR_INPUT

	sInputMessage: STRING(255);
	sFileName: T_MaxString;
	sDirectory: T_MaxString;
	bEnable: BOOL;

END_VAR
VAR_OUTPUT

	sDate: STRING;

	bNewDateFound: BOOL;
END_VAR

VAR_OUTPUT PERSISTENT
	sOldFileName: T_MaxString;
	sFilePathFinal: t_MaxString;
END_VAR
VAR PERSISTENT
	sOldDate: STRING;
	sNewFileName_Temp: T_MaxString;
END_VAR
VAR_IN_OUT PERSISTENT
	wToday: STRING;
END_VAR
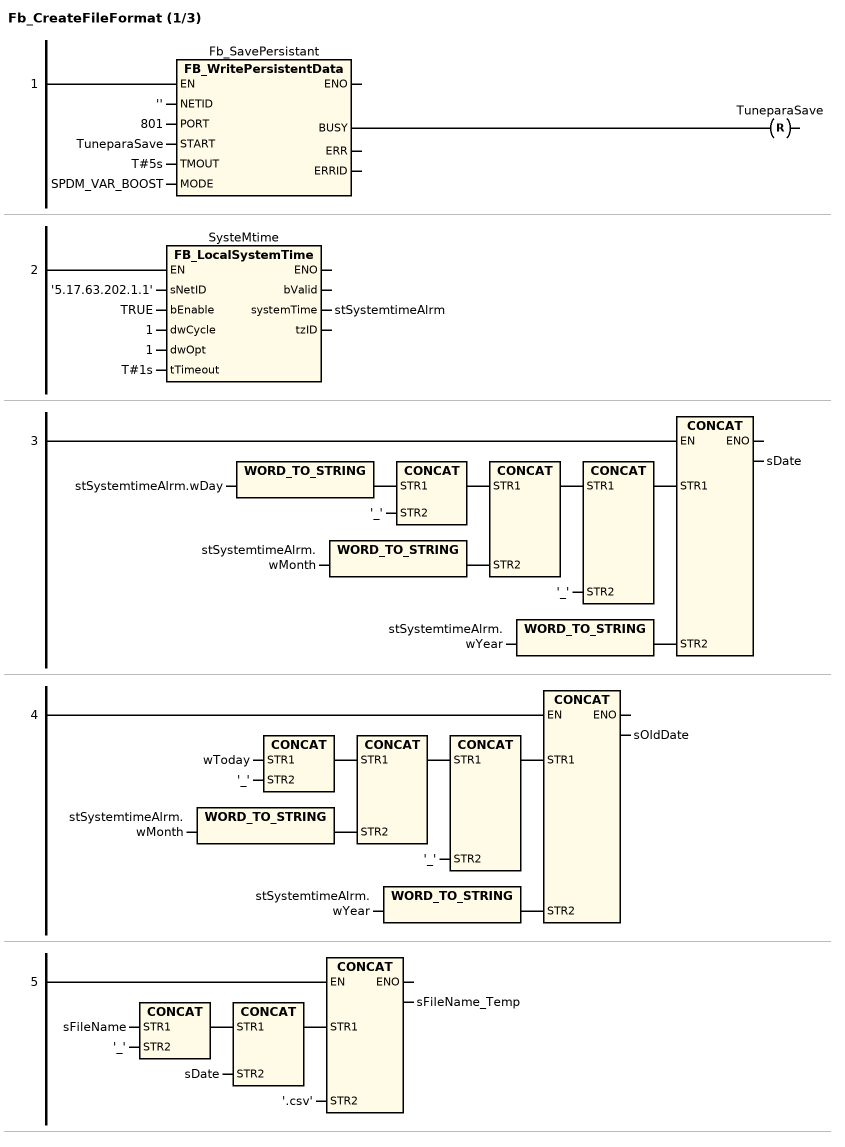
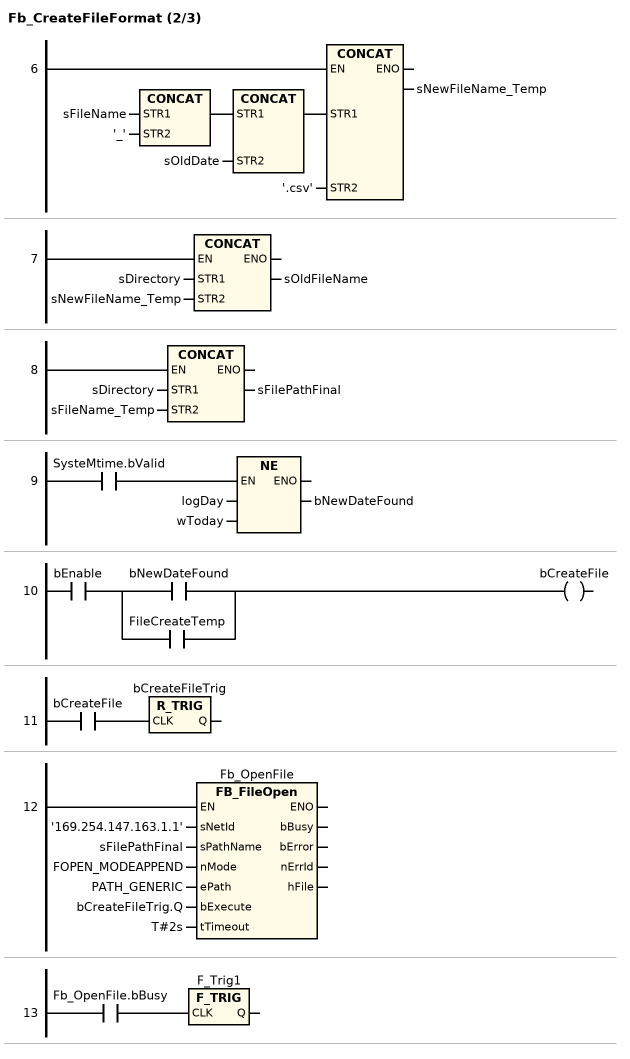
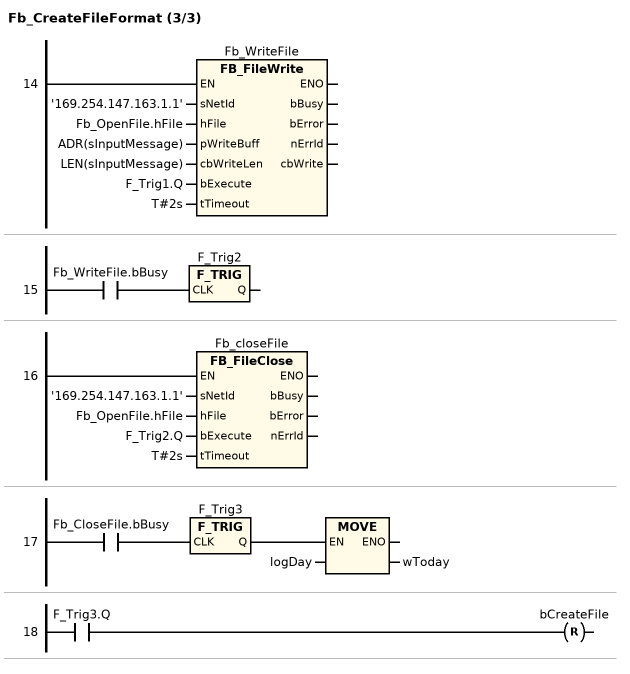
_LD_ (* Ladder Diagram *)
NETWORK 1
	*
		EN --- Fb_SavePersistant:FB_WritePersistentData(NETID: '', PORT: 801, START: TuneparaSave, TMOUT: T#5s, MODE: SPDM_VAR_BOOST) => R TuneparaSave
NETWORK 2
	*
		EN --- SysteMtime:FB_LocalSystemTime(sNetID: '5.17.63.202.1.1', bEnable: TRUE, dwCycle: 1, dwOpt: 1, tTimeout: T#1s, systemTime => stSystemtimeAlrm)
NETWORK 3
	*
		EN --- CONCAT(STR1: CONCAT(STR1: CONCAT(STR1: CONCAT(STR1: WORD_TO_STRING(stSystemtimeAlrm.wDay), STR2: '_'), STR2: WORD_TO_STRING(stSystemtimeAlrm.wMonth)), STR2: '_'), STR2: WORD_TO_STRING(stSystemtimeAlrm.wYear)) => sDate
NETWORK 4
	*
		EN --- CONCAT(STR1: CONCAT(STR1: CONCAT(STR1: CONCAT(STR1: wToday, STR2: '_'), STR2: WORD_TO_STRING(stSystemtimeAlrm.wMonth)), STR2: '_'), STR2: WORD_TO_STRING(stSystemtimeAlrm.wYear)) => sOldDate
NETWORK 5
	*
		EN --- CONCAT(STR1: CONCAT(STR1: CONCAT(STR1: sFileName, STR2: '_'), STR2: sDate), STR2: '.csv') => sFileName_Temp
NETWORK 6
	*
		EN --- CONCAT(STR1: CONCAT(STR1: CONCAT(STR1: sFileName, STR2: '_'), STR2: sOldDate), STR2: '.csv') => sNewFileName_Temp
NETWORK 7
	*
		EN --- CONCAT(STR1: sDirectory, STR2: sNewFileName_Temp) => sOldFileName
NETWORK 8
	*
		EN --- CONCAT(STR1: sDirectory, STR2: sFileName_Temp) => sFilePathFinal
NETWORK 9
	[SysteMtime.bValid]
		EN --- NE(logDay, wToday) => bNewDateFound
NETWORK 10
	[bEnable] - { [bNewDateFound] | [FileCreateTemp] } --- (bCreateFile)
NETWORK 11
	[bCreateFile] - bCreateFileTrig:R_TRIG(CLK: *)
NETWORK 12
	*
		EN --- Fb_OpenFile:FB_FileOpen(sNetId: '169.254.147.163.1.1', sPathName: sFilePathFinal, nMode: FOPEN_MODEAPPEND, ePath: PATH_GENERIC, bExecute: bCreateFileTrig.Q, tTimeout: T#2s)
NETWORK 13
	[Fb_OpenFile.bBusy] - F_Trig1:F_TRIG(CLK: *)
NETWORK 14
	*
		EN --- Fb_WriteFile:FB_FileWrite(sNetId: '169.254.147.163.1.1', hFile: Fb_OpenFile.hFile, pWriteBuff: ADR(sInputMessage), cbWriteLen: LEN(sInputMessage), bExecute: F_Trig1.Q, tTimeout: T#2s)
NETWORK 15
	[Fb_WriteFile.bBusy] - F_Trig2:F_TRIG(CLK: *)
NETWORK 16
	*
		EN --- Fb_closeFile:FB_FileClose(sNetId: '169.254.147.163.1.1', hFile: Fb_OpenFile.hFile, bExecute: F_Trig2.Q, tTimeout: T#2s)
NETWORK 17
	[Fb_CloseFile.bBusy] - F_Trig3:F_TRIG(CLK: *)
		EN --- MOVE(logDay) => wToday
NETWORK 18
	[F_Trig3.Q] --- (R bCreateFile)
_END_LD_
(* the same logic as Structured Text *)
(* Network 1 *)
Fb_SavePersistant(NETID := '', PORT := 801, START := TuneparaSave, TMOUT := T#5s, MODE := SPDM_VAR_BOOST);
IF Fb_SavePersistant.BUSY THEN TuneparaSave := FALSE; END_IF;
(* Network 2 *)
SysteMtime(sNetID := '5.17.63.202.1.1', bEnable := TRUE, dwCycle := 1, dwOpt := 1, tTimeout := T#1s);
stSystemtimeAlrm := SysteMtime.systemTime;
(* Network 3 *)
sDate := CONCAT(CONCAT(CONCAT(CONCAT(WORD_TO_STRING(stSystemtimeAlrm.wDay), '_'), WORD_TO_STRING(stSystemtimeAlrm.wMonth)), '_'), WORD_TO_STRING(stSystemtimeAlrm.wYear));
(* Network 4 *)
sOldDate := CONCAT(CONCAT(CONCAT(CONCAT(wToday, '_'), WORD_TO_STRING(stSystemtimeAlrm.wMonth)), '_'), WORD_TO_STRING(stSystemtimeAlrm.wYear));
(* Network 5 *)
sFileName_Temp := CONCAT(CONCAT(CONCAT(sFileName, '_'), sDate), '.csv');
(* Network 6 *)
sNewFileName_Temp := CONCAT(CONCAT(CONCAT(sFileName, '_'), sOldDate), '.csv');
(* Network 7 *)
sOldFileName := CONCAT(sDirectory, sNewFileName_Temp);
(* Network 8 *)
sFilePathFinal := CONCAT(sDirectory, sFileName_Temp);
(* Network 9 *)
IF SysteMtime.bValid THEN
	bNewDateFound := logDay <> wToday;
END_IF;
(* Network 10 *)
bCreateFile := bEnable AND (bNewDateFound OR FileCreateTemp);
(* Network 11 *)
bCreateFileTrig(CLK := bCreateFile);
(* Network 12 *)
Fb_OpenFile(sNetId := '169.254.147.163.1.1', sPathName := sFilePathFinal, nMode := FOPEN_MODEAPPEND, ePath := PATH_GENERIC, bExecute := bCreateFileTrig.Q, tTimeout := T#2s);
(* Network 13 *)
F_Trig1(CLK := Fb_OpenFile.bBusy);
(* Network 14 *)
Fb_WriteFile(sNetId := '169.254.147.163.1.1', hFile := Fb_OpenFile.hFile, pWriteBuff := ADR(sInputMessage), cbWriteLen := LEN(sInputMessage), bExecute := F_Trig1.Q, tTimeout := T#2s);
(* Network 15 *)
F_Trig2(CLK := Fb_WriteFile.bBusy);
(* Network 16 *)
Fb_closeFile(sNetId := '169.254.147.163.1.1', hFile := Fb_OpenFile.hFile, bExecute := F_Trig2.Q, tTimeout := T#2s);
(* Network 17 *)
F_Trig3(CLK := Fb_CloseFile.bBusy);
IF F_Trig3.Q THEN
	wToday := logDay;
END_IF;
(* Network 18 *)
IF F_Trig3.Q THEN bCreateFile := FALSE; END_IF;
END_FUNCTION_BLOCK

(* POU FunctionBlocks/Fb_FormatDrive, FBD *)
FUNCTION_BLOCK Fb_FormatDrive
VAR_INPUT
	sDriveName: T_MaxString;
	bFormatDisk: BOOL;
END_VAR
VAR_OUTPUT
END_VAR
VAR
	sDeleteCommand_Temp: T_MaxString;
	sDeleteCommand: T_MaxString;
	nDirectoryLength: INT;
	sFormatedDirectory: T_MaxString;
	FbFormatDisk: NT_StartProcess;
END_VAR
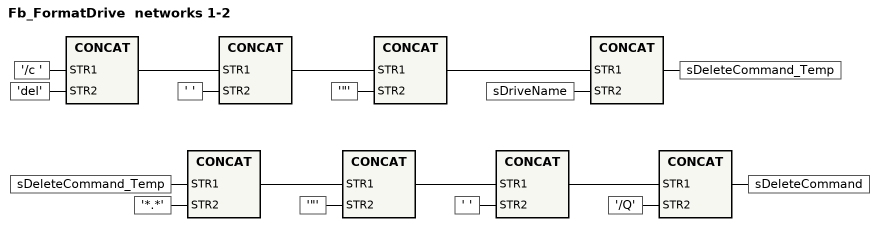
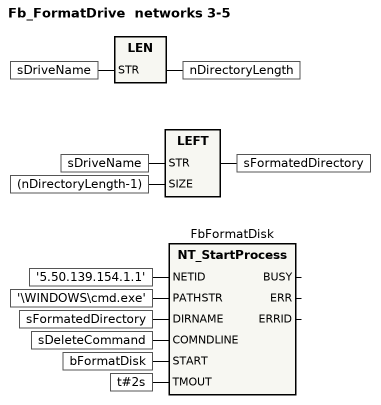
_FBD_ (* Function Block Diagram *)
NETWORK 1
	CONCAT(STR1: CONCAT(STR1: CONCAT(STR1: CONCAT(STR1: '/c ', STR2: 'del'), STR2: ' '), STR2: '"'), STR2: sDriveName) => sDeleteCommand_Temp
NETWORK 2
	CONCAT(STR1: CONCAT(STR1: CONCAT(STR1: CONCAT(STR1: sDeleteCommand_Temp, STR2: '*.*'), STR2: '"'), STR2: ' '), STR2: '/Q') => sDeleteCommand
NETWORK 3
	LEN(STR: sDriveName) => nDirectoryLength
NETWORK 4
	LEFT(STR: sDriveName, SIZE: (nDirectoryLength-1)) => sFormatedDirectory
NETWORK 5
	FbFormatDisk:NT_StartProcess(NETID: '5.50.139.154.1.1', PATHSTR: '\WINDOWS\cmd.exe', DIRNAME: sFormatedDirectory, COMNDLINE: sDeleteCommand, START: bFormatDisk, TMOUT: t#2s)
_END_FBD_
(* the same logic as Structured Text *)
(* Network 1 *)
sDeleteCommand_Temp := CONCAT(CONCAT(CONCAT(CONCAT('/c ', 'del'), ' '), '"'), sDriveName);
(* Network 2 *)
sDeleteCommand := CONCAT(CONCAT(CONCAT(CONCAT(sDeleteCommand_Temp, '*.*'), '"'), ' '), '/Q');
(* Network 3 *)
nDirectoryLength := LEN(sDriveName);
(* Network 4 *)
sFormatedDirectory := LEFT(sDriveName, (nDirectoryLength-1));
(* Network 5 *)
FbFormatDisk(NETID := '5.50.139.154.1.1', PATHSTR := '\WINDOWS\cmd.exe', DIRNAME := sFormatedDirectory, COMNDLINE := sDeleteCommand, START := bFormatDisk, TMOUT := t#2s);
END_FUNCTION_BLOCK

(* POU FunctionBlocks/Fb_CopyFileToRemotePC, FBD *)
FUNCTION_BLOCK Fb_CopyFileToRemotePC
VAR
	sCopyFileCommandTemp: T_MaxString;
	sFormatedDestDirectory: T_Maxstring;
	sCopyFileCommand: T_MaxString;
	sFormatedDirectory: T_MaxString;
	sMakeDirCommand: T_MaxString;

	Fb_SystemTime: FB_LocalSystemTime;
	FB_MakeDirectory: NT_StartProcess;
	Fb_CopyFiles: NT_StartProcess;
END_VAR
VAR_INPUT

	bMakeDirectory: BOOL;
	bCopyFile: BOOL;
	sDestDriveName: T_MaxString;
	sSourceDirectory: T_MaxString;
END_VAR
VAR_OUTPUT
	sFinalDestDirectory: T_MaxString;
END_VAR
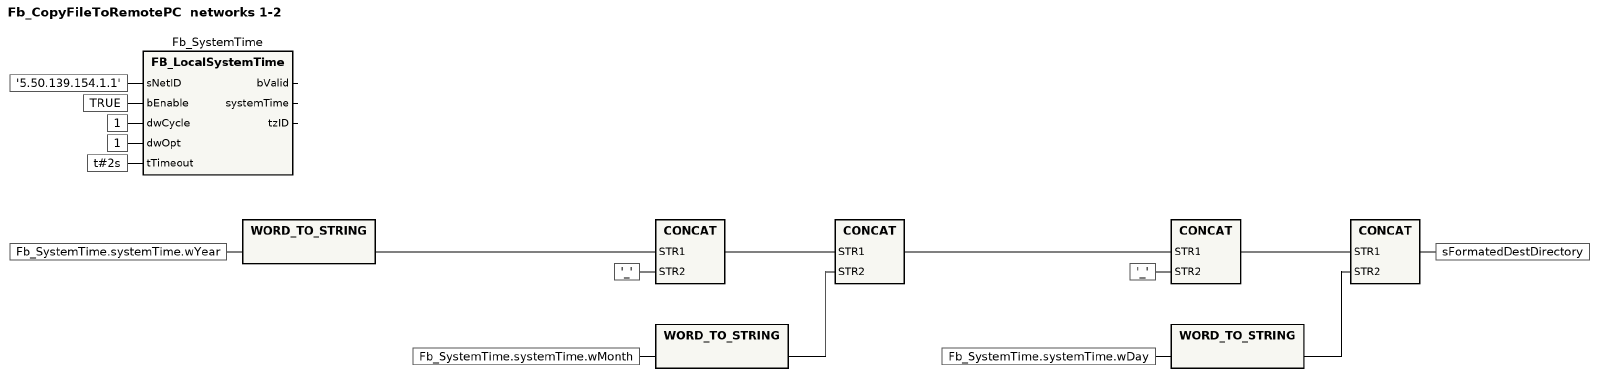
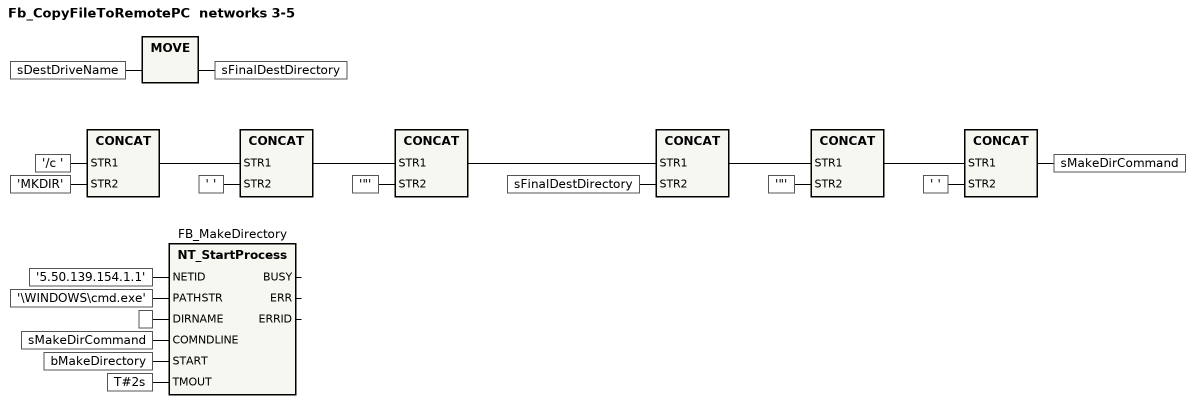
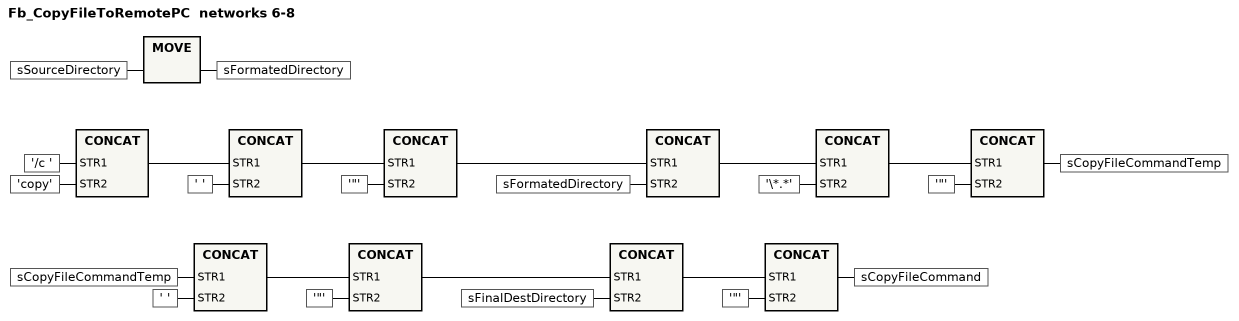
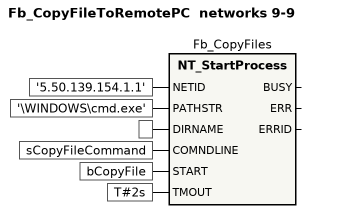
_FBD_ (* Function Block Diagram *)
NETWORK 1
	Fb_SystemTime:FB_LocalSystemTime(sNetID: '5.50.139.154.1.1', bEnable: TRUE, dwCycle: 1, dwOpt: 1, tTimeout: t#2s)
NETWORK 2
	CONCAT(STR1: CONCAT(STR1: CONCAT(STR1: CONCAT(STR1: WORD_TO_STRING(Fb_SystemTime.systemTime.wYear), STR2: '_'), STR2: WORD_TO_STRING(Fb_SystemTime.systemTime.wMonth)), STR2: '_'), STR2: WORD_TO_STRING(Fb_SystemTime.systemTime.wDay)) => sFormatedDestDirectory
NETWORK 3
	MOVE(sDestDriveName) => sFinalDestDirectory
NETWORK 4
	CONCAT(STR1: CONCAT(STR1: CONCAT(STR1: CONCAT(STR1: CONCAT(STR1: CONCAT(STR1: '/c ', STR2: 'MKDIR'), STR2: ' '), STR2: '"'), STR2: sFinalDestDirectory), STR2: '"'), STR2: ' ') => sMakeDirCommand
NETWORK 5
	FB_MakeDirectory:NT_StartProcess(NETID: '5.50.139.154.1.1', PATHSTR: '\WINDOWS\cmd.exe', DIRNAME: , COMNDLINE: sMakeDirCommand, START: bMakeDirectory, TMOUT: T#2s)
NETWORK 6
	MOVE(sSourceDirectory) => sFormatedDirectory
NETWORK 7
	CONCAT(STR1: CONCAT(STR1: CONCAT(STR1: CONCAT(STR1: CONCAT(STR1: CONCAT(STR1: '/c ', STR2: 'copy'), STR2: ' '), STR2: '"'), STR2: sFormatedDirectory), STR2: '\*.*'), STR2: '"') => sCopyFileCommandTemp
NETWORK 8
	CONCAT(STR1: CONCAT(STR1: CONCAT(STR1: CONCAT(STR1: sCopyFileCommandTemp, STR2: ' '), STR2: '"'), STR2: sFinalDestDirectory), STR2: '"') => sCopyFileCommand
NETWORK 9
	Fb_CopyFiles:NT_StartProcess(NETID: '5.50.139.154.1.1', PATHSTR: '\WINDOWS\cmd.exe', DIRNAME: , COMNDLINE: sCopyFileCommand, START: bCopyFile, TMOUT: T#2s)
_END_FBD_
(* the same logic as Structured Text *)
(* Network 1 *)
Fb_SystemTime(sNetID := '5.50.139.154.1.1', bEnable := TRUE, dwCycle := 1, dwOpt := 1, tTimeout := t#2s);
(* Network 2 *)
sFormatedDestDirectory := CONCAT(CONCAT(CONCAT(CONCAT(WORD_TO_STRING(Fb_SystemTime.systemTime.wYear), '_'), WORD_TO_STRING(Fb_SystemTime.systemTime.wMonth)), '_'), WORD_TO_STRING(Fb_SystemTime.systemTime.wDay));
(* Network 3 *)
sFinalDestDirectory := sDestDriveName;
(* Network 4 *)
sMakeDirCommand := CONCAT(CONCAT(CONCAT(CONCAT(CONCAT(CONCAT('/c ', 'MKDIR'), ' '), '"'), sFinalDestDirectory), '"'), ' ');
(* Network 5: see the listing above *)
(* Network 6 *)
sFormatedDirectory := sSourceDirectory;
(* Network 7 *)
sCopyFileCommandTemp := CONCAT(CONCAT(CONCAT(CONCAT(CONCAT(CONCAT('/c ', 'copy'), ' '), '"'), sFormatedDirectory), '\*.*'), '"');
(* Network 8 *)
sCopyFileCommand := CONCAT(CONCAT(CONCAT(CONCAT(sCopyFileCommandTemp, ' '), '"'), sFinalDestDirectory), '"');
(* Network 9: see the listing above *)
END_FUNCTION_BLOCK

(* POU Auto1/DataLog/DataLog_Alarm, ST *)
PROGRAM DataLog_Alarm
VAR
	stStation1_ProductionData: Production_Data;
	ST1_ProductionDataValues: STRING(3000);
	S1_iCyc_Count_DISP: INT;
	S1_iACT_HLD_TIMEDISP: INT;
	stActiveuserCredential: BOOL;
	nPressureMaxvalue: REAL;
	OperatorName: STRING;
	nMinimumTopTempLimit_ST1: INT;
	nMaximumTopTempLimit_ST1: INT;
	nTOPTempMaxvalue: UINT;
	nMinimumBTMTempLimit_ST1: INT;
	nBTMTempMaxvalue: UINT;
	nMaximumBTMTempLimit_ST1: INT;
	Set_HLDTIME: INT;
	S_1_iPressure: REAL;
	rS_PressureRange1: REAL;
	nMaxEnergy: REAL;
	nMaxPower: REAL;
	S_iSET_COUNT: INT;
	S1_iTotCyc_Count_DISP: INT;
	sJobStatus_ST1: STRING;
	sStation1_ProductionData_FileName: STRING(80) := 'Hard Disk\Reports\Test1\ProductionData.csv';
	Fb_LoagProductionData: DATA_LOG_Save;
	SaveData: BOOL;
	ST1_ProductionData: STRING(500);
	Fb_CreateFileFormat_1: Fb_CreateFileFormat;
	bEnableFileFormat: BOOL;
	wTodayTemp: STRING;
	sDateTemp: STRING;
	sOLDFileName_ST1: T_MaxString;
	Fb_FormatDrive_1: Fb_FormatDrive;
	bFileDelete: BOOL;
	Fb_CopyBackupAL_Server_LogOf_1: Fb_CopyFileToRemotePC;
	bool2: BOOL;
	bAstart: BOOL;
	TON_1: TON;
	TON_2: TON;
	CTU_1: CTU;
	R_TRIG_1: R_TRIG;
	R_TRIG_2: R_TRIG;
	bACreateNewFile: BOOL;
	ReportStep: INT;
	bANewDay: BOOL;
	Timer1: TON;
	Timer2: TON;
	R_TRIG1: R_TRIG;


	iUnitBNetWtTemp1: REAL;
	rRetUnitBWeightTemp1: REAL;
	StepTemp1: INT;
	rRetUnitBWeightTemp2: REAL;
	StepTemp2: INT;
	BCreateDir: BOOL;
	FB_CreateDir_1: FB_CreateDir;
	bANewDaytemp: BOOL;
	bit2: BOOL;
	hfile: UINT;
	FB_FileOpen_1: FB_FileOpen;
	test: BOOL;
	bit3: BOOL;
	FB_FileWrite_1: FB_FileWrite;
	bEnableFileFormattemp: BOOL;
	BDelete: BOOL;
	FB_FileDelete_1: FB_FileDelete;
	Timer3: TON;
	iCartoNoHmiTemp: DWORD;
	dateInint: WORD;
	Fb_CreateFileFormat_Alarm: Fb_CreateFileFormat_Alarm;
	ST1_ErrorAlarmData: STRING(500);
	stStation1_ErrorAlarmData: ErrorAlarm_Data;
	ST1_ErrorAlarmDataValues: STRING(3000);
	sStation1_ErrorAlarmData_FileName: STRING;
	Fb_LoagErrorAlarmData: AlarmErrorDATA_LOG_Save;


	bFileDelete_1: BOOL;
	E_OpenPath: E_OpenPath;
END_VAR
FileCreateTemp;

Fb_CreateFileFormat_Alarm(
	sInputMessage:=ST1_ErrorAlarmData ,
	sFileName:='ErrorAlarmData' ,
	sDirectory:= '\\NITINK2-PC\Report\' (*  'Hard Disk\Reports\Indo\'  *) ,
	bEnable:=bEnableFileFormat ,
	wToday:=wTodayTemp ,
	sDate=> sDateTemp,
	bNewDateFound=> bANewDay,
	sOldFileName=>sOLDFileName_ST1 ,
	sFilePathFinal=> );

FB_FileDelete_1(
	sNetId:='124.124.124.197.1.1' ,
	sPathName:= sStation1_ErrorAlarmData_FileName ,
	ePath:=E_OpenPath ,
	bExecute:=bFileDelete_1 ,
	tTimeout:=t#1s ,
	bBusy=> ,
	bError=> ,
	nErrId=> );


	stStation1_ErrorAlarmData.Error_No							:=(* INT_TO_STRING*)( AlarmBitArray );
	stStation1_ErrorAlarmData.SDateF							:= (wTodayToHmi);
	stStation1_ErrorAlarmData.sShift								:=(sShitToReport);
	stStation1_ErrorAlarmData.Time_No							:=(sTIME);



							(*	######## LOG PRODUCTION DATA		#####	*)


	ST1_ErrorAlarmDataValues:= CONCAT(stStation1_ErrorAlarmData.Error_No,',');
	ST1_ErrorAlarmDataValues:=	 CONCAT( ST1_ErrorAlarmDataValues,stStation1_ErrorAlarmData.SDateF);
	ST1_ErrorAlarmDataValues:= CONCAT( ST1_ErrorAlarmDataValues,',');
	ST1_ErrorAlarmDataValues:=	 CONCAT( ST1_ErrorAlarmDataValues,stStation1_ErrorAlarmData.sShift	);
	ST1_ErrorAlarmDataValues:= CONCAT( ST1_ErrorAlarmDataValues,',');
	ST1_ErrorAlarmDataValues:=	 CONCAT( ST1_ErrorAlarmDataValues,stStation1_ErrorAlarmData.Time_No	);
	ST1_ErrorAlarmDataValues:= CONCAT( ST1_ErrorAlarmDataValues,'$0A');


									(*==========Saving the Data to Report===========*)

sStation1_ErrorAlarmData_FileName:= Fb_CreateFileFormat_Alarm.sOldFileName ;    (*    'Hard Disk\Reports\Test1\ProductionData.csv' ;*)


Fb_LoagErrorAlarmData(
	bStartDataLog:= SaveData ,
	sDataLogFileName:=sStation1_ErrorAlarmData_FileName ,
	LogData:=ST1_ErrorAlarmDataValues ,
	bErrorDataLog=> );


			(*=============== file copy from CX Controller to Remote PC & File Delete In CX Device======================*)


	Fb_CopyBackupAL_Server_LogOf_1(
		bMakeDirectory:= ,
		bCopyFile:=bool2,
		sDestDriveName:= '\\NITINK2-PC\Report\' ,
		sSourceDirectory:='\Hard Disk\Reports\Indo' ,
		 );


(*
Fb_FormatDrive_1(sDriveName:='\\WELCOME-PC\Reports\' , bFormatDisk:=bFileDelete );*)


CASE ReportStep OF

	0:	 IF R_TRIG1.Q   THEN FileCreateTemp:=TRUE; Timer3(IN:=FALSE); ReportStep:=1; END_IF

	1:	(*		##### Station 1 Production Data	#####	*)

		ST1_ErrorAlarmData:= CONCAT( 'Error No',',');
		ST1_ErrorAlarmData:=	 CONCAT( ST1_ErrorAlarmData,'Date');
		ST1_ErrorAlarmData:= CONCAT( ST1_ErrorAlarmData,',');
		ST1_ErrorAlarmData:=	 CONCAT( ST1_ErrorAlarmData,'Shift');
		ST1_ErrorAlarmData:= CONCAT( ST1_ErrorAlarmData,',');
		ST1_ErrorAlarmData:=	 CONCAT( ST1_ErrorAlarmData,'Time');
		ST1_ErrorAlarmData:= CONCAT( ST1_ErrorAlarmData,'$0A');

		ReportStep:=2;

	2:	Timer1(IN:=FALSE);
		bANewDay:=FALSE;
		ReportStep:=3;


	3:	bEnableFileFormat:=TRUE;
		Timer1(IN:=TRUE , PT:=T#100ms , Q=> , ET=> );
		IF Timer1.Q THEN bEnableFileFormat:=FALSE;  ReportStep:=4; END_IF


	4:	(*IF R_TRIG1.Q THEN  *)
		SaveData:=TRUE;
		Timer1(IN:=FALSE);
		ReportStep:=5;

	5:	Timer3(IN:=TRUE , PT:=T#5s , Q=> , ET=> );
		IF Timer3.Q THEN SaveData:=FALSE; bFileDelete_1:=TRUE;  ReportStep:=6; END_IF

	6:	 bFileDelete_1:=FALSE;Timer3(IN:=FALSE); FileCreateTemp:=FALSE; ReportStep:=0;

END_CASE



R_TRIG1(CLK:=ERROR_ALERT , Q=> );



IF bASupplyPressureError 										THEN AlarmBitArray :='1' ; END_IF
IF bAConeFeddCylFwdRsError									THEN AlarmBitArray :='2' ; END_IF
IF bAWrap_1PistRsError										THEN AlarmBitArray :='3 '; END_IF
IF bAWrap_2PistRsError									    	THEN AlarmBitArray:='4' ; END_IF
IF bAWrap_3PistRsError										THEN AlarmBitArray :='5' ; END_IF
IF bAForwPistRsError											THEN AlarmBitArray :='6' ; END_IF

IF bASealBottomRsError			     							THEN AlarmBitArray :='7' ; END_IF
IF bASealTopPistRsError										THEN AlarmBitArray :='8' ; END_IF
IF bASealSepaX_axisRsError									THEN AlarmBitArray :='9' ; END_IF
IF bASealSepaY_axisRsError									THEN AlarmBitArray :='10' ; END_IF
IF bATiltPistRsError											THEN AlarmBitArray:='11' ; END_IF
IF bAReversPistnRsError										THEN AlarmBitArray := '12'; END_IF

IF bAColumnPushPistnRsError									THEN AlarmBitArray :='13' ; END_IF
IF bAConeEjectPistnRsError									THEN AlarmBitArray :='14' ; END_IF
IF bASepaHoriForwdEndRsError								THEN AlarmBitArray :='15' ; END_IF
IF bASepaVertiEndPistnRsError									THEN AlarmBitArray :='16' ; END_IF
IF bASepaVerCylhomeRsError									THEN AlarmBitArray :='17' ; END_IF
IF bASepaHoriRevValveRsError									THEN AlarmBitArray :='18' ; END_IF

IF bAL_BTightHomeSenRsError									THEN AlarmBitArray :='19' ; END_IF
IF bAGrossWtSenRsError										THEN AlarmBitArray :='20' ; END_IF
IF bAGrossWtHomeSenRsError									THEN AlarmBitArray := '21'; END_IF
IF bACartonSenRsError										THEN AlarmBitArray :='22' ; END_IF
IF bARowStoppHomeSenRsError								THEN AlarmBitArray :='23' ; END_IF
IF bAConeOnMatrixConv										THEN AlarmBitArray :='24'; END_IF


IF bGrossWieghtNOk											THEN AlarmBitArray :='25 '; END_IF
IF bSealConveyerConePresent									THEN AlarmBitArray :='26' ; END_IF
IF bEmptyCartonDetectError										THEN AlarmBitArray :='27'; END_IF
IF bAConeMissErrorAtWrpConv									THEN AlarmBitArray :='28' ; END_IF
IF bACheckWrappConv										THEN AlarmBitArray :='29' ; END_IF
IF bHmiColourChangeBit2_24									THEN AlarmBitArray :='30'; END_IF



IF bAPolythinSheetError										THEN AlarmBitArray :='31' ; END_IF
IF bAConeMissAtMatricConv									THEN AlarmBitArray :='32' ; END_IF
IF SeparatorAlertbit											THEN AlarmBitArray :='33'; END_IF  (* Sensor Error in Carton Conveyor*)
IF SealBitAlert												THEN AlarmBitArray :='34' ; END_IF
(*IF bAConeMissAtMatricConv								THEN AlarmBitArray :='35' ; END_IF
IF bHmiColourChangeBit									THEN AlarmBitArray :='36'; END_IF  (*Clear Carton at full Carton Conveyor*)


IF SeparatorAlertbit										THEN AlarmBitArray :='37 '; END_IF
(*IF bAGrossWtSenRsError									THEN AlarmBitArray :='38' ; END_IF
IF bAGrossWtHomeSenRsError								THEN AlarmBitArray :='39'; END_IF
IF bACartonSenRsError									THEN AlarmBitArray :='40' ; END_IF
IF bARowStoppHomeSenRsError							THEN AlarmBitArray :='41' ; END_IF
IF bAConeOnMatrixConv									THEN AlarmBitArray :='42'; END_IF *)
*)
END_PROGRAM

(* POU FunctionBlocks/Fb_CreateFileFormat_Alarm, LD *)
FUNCTION_BLOCK Fb_CreateFileFormat_Alarm
VAR
	Fb_OpenFile: FB_FileOpen;
	Fb_WriteFile: FB_FileWrite;
	F_Trig1: F_TRIG;
	F_Trig2: F_TRIG;
	Fb_closeFile: FB_FileClose;
	F_Trig3: F_TRIG;


	SysteMtime: FB_LocalSystemTime;
	stSystemtimeAlrm: Timestruct;

	sFileName_Temp: T_MaxString;


	bCreateFileTrig: R_TRIG;
	bCreateFile: BOOL;
	Fb_SavePersistant: FB_WritePersistentData;
	TuneparaSave: BOOL;
END_VAR
VAR_INPUT

	sInputMessage: STRING(255);
	sFileName: T_MaxString;
	sDirectory: T_MaxString;
	bEnable: BOOL;

END_VAR
VAR_OUTPUT

	sDate: STRING;

	bNewDateFound: BOOL;
END_VAR

VAR_OUTPUT PERSISTENT
	sOldFileName: T_MaxString;
	sFilePathFinal: t_MaxString;
END_VAR
VAR PERSISTENT
	sOldDate: STRING;
	sNewFileName_Temp: T_MaxString;
END_VAR
VAR_IN_OUT PERSISTENT
	wToday: STRING;
END_VAR
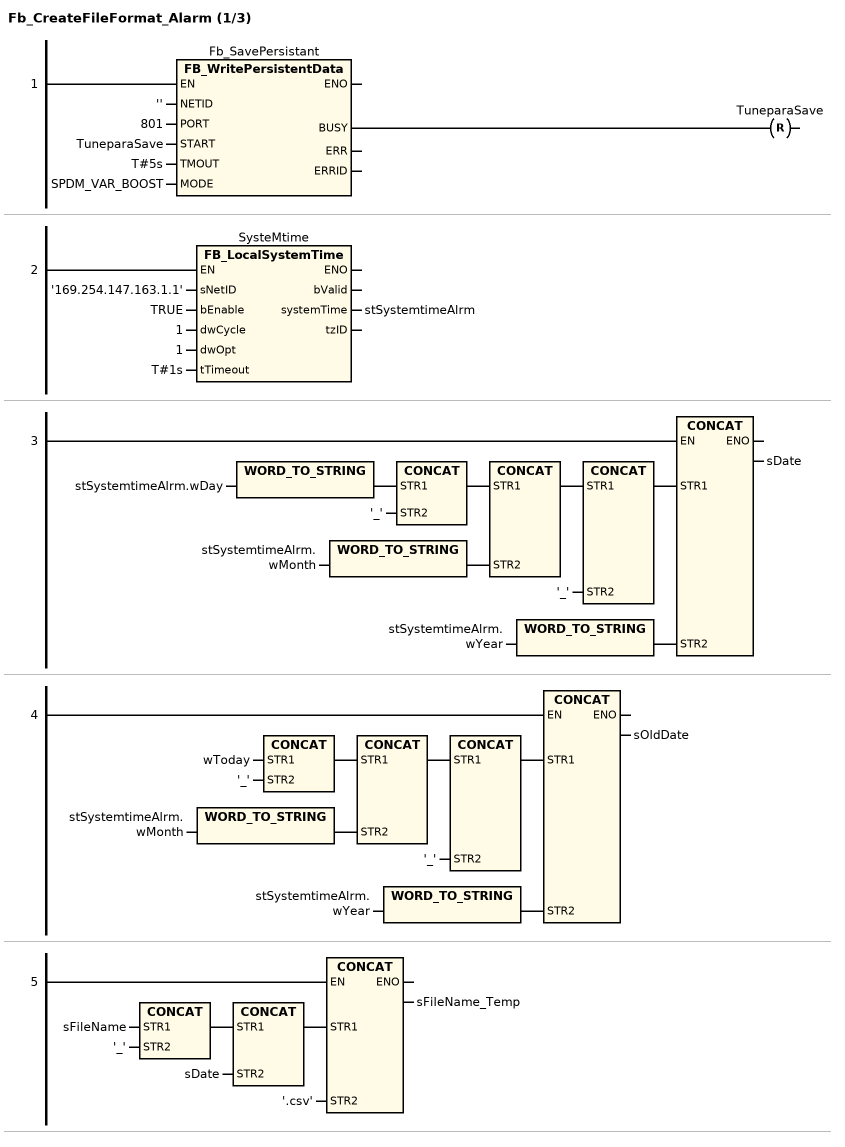
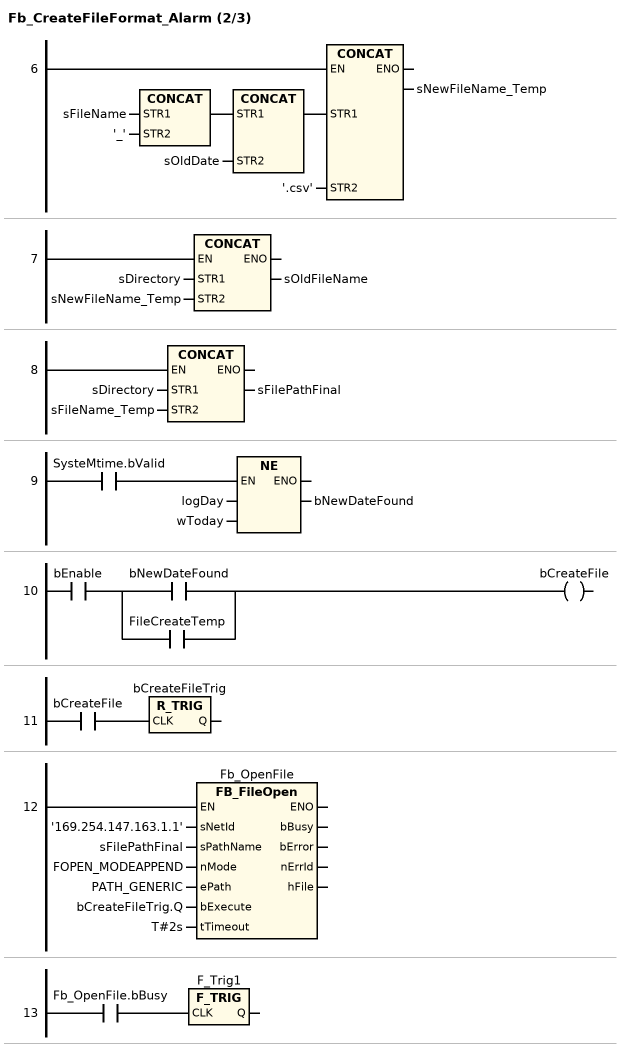
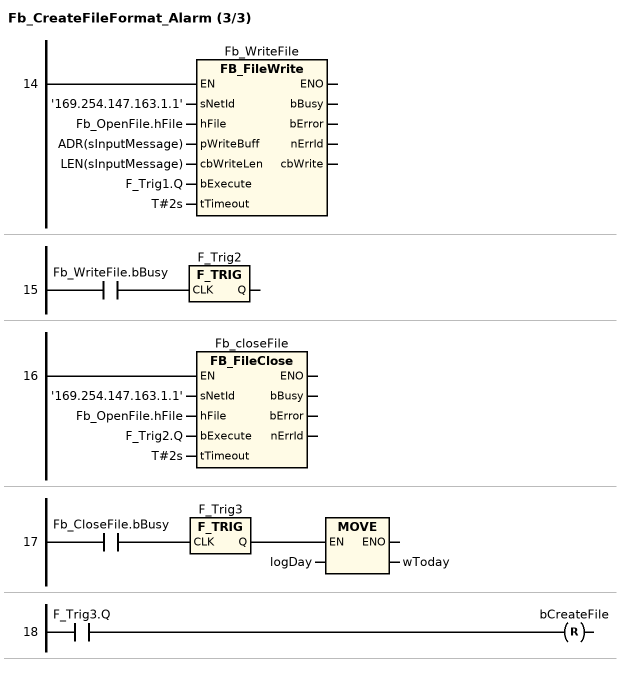
_LD_ (* Ladder Diagram *)
NETWORK 1
	*
		EN --- Fb_SavePersistant:FB_WritePersistentData(NETID: '', PORT: 801, START: TuneparaSave, TMOUT: T#5s, MODE: SPDM_VAR_BOOST) => R TuneparaSave
NETWORK 2
	*
		EN --- SysteMtime:FB_LocalSystemTime(sNetID: '169.254.147.163.1.1', bEnable: TRUE, dwCycle: 1, dwOpt: 1, tTimeout: T#1s, systemTime => stSystemtimeAlrm)
NETWORK 3
	*
		EN --- CONCAT(STR1: CONCAT(STR1: CONCAT(STR1: CONCAT(STR1: WORD_TO_STRING(stSystemtimeAlrm.wDay), STR2: '_'), STR2: WORD_TO_STRING(stSystemtimeAlrm.wMonth)), STR2: '_'), STR2: WORD_TO_STRING(stSystemtimeAlrm.wYear)) => sDate
NETWORK 4
	*
		EN --- CONCAT(STR1: CONCAT(STR1: CONCAT(STR1: CONCAT(STR1: wToday, STR2: '_'), STR2: WORD_TO_STRING(stSystemtimeAlrm.wMonth)), STR2: '_'), STR2: WORD_TO_STRING(stSystemtimeAlrm.wYear)) => sOldDate
NETWORK 5
	*
		EN --- CONCAT(STR1: CONCAT(STR1: CONCAT(STR1: sFileName, STR2: '_'), STR2: sDate), STR2: '.csv') => sFileName_Temp
NETWORK 6
	*
		EN --- CONCAT(STR1: CONCAT(STR1: CONCAT(STR1: sFileName, STR2: '_'), STR2: sOldDate), STR2: '.csv') => sNewFileName_Temp
NETWORK 7
	*
		EN --- CONCAT(STR1: sDirectory, STR2: sNewFileName_Temp) => sOldFileName
NETWORK 8
	*
		EN --- CONCAT(STR1: sDirectory, STR2: sFileName_Temp) => sFilePathFinal
NETWORK 9
	[SysteMtime.bValid]
		EN --- NE(logDay, wToday) => bNewDateFound
NETWORK 10
	[bEnable] - { [bNewDateFound] | [FileCreateTemp] } --- (bCreateFile)
NETWORK 11
	[bCreateFile] - bCreateFileTrig:R_TRIG(CLK: *)
NETWORK 12
	*
		EN --- Fb_OpenFile:FB_FileOpen(sNetId: '169.254.147.163.1.1', sPathName: sFilePathFinal, nMode: FOPEN_MODEAPPEND, ePath: PATH_GENERIC, bExecute: bCreateFileTrig.Q, tTimeout: T#2s)
NETWORK 13
	[Fb_OpenFile.bBusy] - F_Trig1:F_TRIG(CLK: *)
NETWORK 14
	*
		EN --- Fb_WriteFile:FB_FileWrite(sNetId: '169.254.147.163.1.1', hFile: Fb_OpenFile.hFile, pWriteBuff: ADR(sInputMessage), cbWriteLen: LEN(sInputMessage), bExecute: F_Trig1.Q, tTimeout: T#2s)
NETWORK 15
	[Fb_WriteFile.bBusy] - F_Trig2:F_TRIG(CLK: *)
NETWORK 16
	*
		EN --- Fb_closeFile:FB_FileClose(sNetId: '169.254.147.163.1.1', hFile: Fb_OpenFile.hFile, bExecute: F_Trig2.Q, tTimeout: T#2s)
NETWORK 17
	[Fb_CloseFile.bBusy] - F_Trig3:F_TRIG(CLK: *)
		EN --- MOVE(logDay) => wToday
NETWORK 18
	[F_Trig3.Q] --- (R bCreateFile)
_END_LD_
(* the same logic as Structured Text *)
(* Network 1 *)
Fb_SavePersistant(NETID := '', PORT := 801, START := TuneparaSave, TMOUT := T#5s, MODE := SPDM_VAR_BOOST);
IF Fb_SavePersistant.BUSY THEN TuneparaSave := FALSE; END_IF;
(* Network 2 *)
SysteMtime(sNetID := '169.254.147.163.1.1', bEnable := TRUE, dwCycle := 1, dwOpt := 1, tTimeout := T#1s);
stSystemtimeAlrm := SysteMtime.systemTime;
(* Network 3 *)
sDate := CONCAT(CONCAT(CONCAT(CONCAT(WORD_TO_STRING(stSystemtimeAlrm.wDay), '_'), WORD_TO_STRING(stSystemtimeAlrm.wMonth)), '_'), WORD_TO_STRING(stSystemtimeAlrm.wYear));
(* Network 4 *)
sOldDate := CONCAT(CONCAT(CONCAT(CONCAT(wToday, '_'), WORD_TO_STRING(stSystemtimeAlrm.wMonth)), '_'), WORD_TO_STRING(stSystemtimeAlrm.wYear));
(* Network 5 *)
sFileName_Temp := CONCAT(CONCAT(CONCAT(sFileName, '_'), sDate), '.csv');
(* Network 6 *)
sNewFileName_Temp := CONCAT(CONCAT(CONCAT(sFileName, '_'), sOldDate), '.csv');
(* Network 7 *)
sOldFileName := CONCAT(sDirectory, sNewFileName_Temp);
(* Network 8 *)
sFilePathFinal := CONCAT(sDirectory, sFileName_Temp);
(* Network 9 *)
IF SysteMtime.bValid THEN
	bNewDateFound := logDay <> wToday;
END_IF;
(* Network 10 *)
bCreateFile := bEnable AND (bNewDateFound OR FileCreateTemp);
(* Network 11 *)
bCreateFileTrig(CLK := bCreateFile);
(* Network 12 *)
Fb_OpenFile(sNetId := '169.254.147.163.1.1', sPathName := sFilePathFinal, nMode := FOPEN_MODEAPPEND, ePath := PATH_GENERIC, bExecute := bCreateFileTrig.Q, tTimeout := T#2s);
(* Network 13 *)
F_Trig1(CLK := Fb_OpenFile.bBusy);
(* Network 14 *)
Fb_WriteFile(sNetId := '169.254.147.163.1.1', hFile := Fb_OpenFile.hFile, pWriteBuff := ADR(sInputMessage), cbWriteLen := LEN(sInputMessage), bExecute := F_Trig1.Q, tTimeout := T#2s);
(* Network 15 *)
F_Trig2(CLK := Fb_WriteFile.bBusy);
(* Network 16 *)
Fb_closeFile(sNetId := '169.254.147.163.1.1', hFile := Fb_OpenFile.hFile, bExecute := F_Trig2.Q, tTimeout := T#2s);
(* Network 17 *)
F_Trig3(CLK := Fb_CloseFile.bBusy);
IF F_Trig3.Q THEN
	wToday := logDay;
END_IF;
(* Network 18 *)
IF F_Trig3.Q THEN bCreateFile := FALSE; END_IF;
END_FUNCTION_BLOCK

(* POU FunctionBlocks/AlarmErrorDATA_LOG_Save, ST *)
FUNCTION_BLOCK AlarmErrorDATA_LOG_Save
VAR_INPUT
	bStartDataLog: BOOL;
	sDataLogFileName: STRING;
	LogData: STRING(1024);

END_VAR
VAR_OUTPUT

	bErrorDataLog: BOOL;
END_VAR
VAR

	R_TRIGStartDataLog: R_TRIG;
	nstep: INT;

	FB_OpenFile_Datalog: FB_FileOpen;
	nFB_OpenFile_Datalog_Errid: UDINT;

	FB_WriteFile_Datalog: FB_FileWrite;
	nFB_WriteFile_Datalog_ErrId: UDINT;

	FB_CloseFile_Datalog: FB_FileClose;
	nFB_CloseFile_Datalog_ErrId: UDINT;
	hDataLogSrcFile: UINT;

END_VAR
R_TRIGStartDataLog(CLK:=bStartDataLog , Q=> );
IF R_TRIGStartDataLog.Q THEN
		nstep :=1;
	END_IF

CASE nstep OF

	0:
		;
		FB_OpenFile_Datalog.bExecute:=FALSE;
		FB_WriteFile_Datalog.bExecute:=FALSE;
		FB_CloseFile_Datalog.bExecute:=FALSE;

	1:(* do nothing *)
		nstep:=nstep+1;

	2:	(* ####	File Open ####*)

			FB_OpenFile_Datalog(  bExecute := FALSE  );
			FB_OpenFile_Datalog(	sNetId :='169.254.147.163.1.1' ,
			sPathName := sDataLogFileName,
			nMode := FOPEN_MODEAPPEND    ,
			ePath := PATH_GENERIC,
			tTimeout := T#2s,
			bExecute := TRUE );
			nstep := nstep+ 1;



	3:		FB_OpenFile_Datalog( bExecute := FALSE );
			IF ( NOT FB_OpenFile_Datalog.bBusy ) THEN
			IF ( FB_OpenFile_Datalog.bError ) THEN
			nFB_OpenFile_Datalog_Errid := FB_OpenFile_Datalog.nErrId;
			bErrorDataLog := TRUE;
			nstep := 50;
			ELSE
			hDataLogSrcFile := FB_OpenFile_Datalog.hFile;
			nstep := nstep + 1;
			END_IF
			END_IF

	4:(*write data to destination file*)
		(*num:=num+1;*)
			FB_WriteFile_Datalog( bExecute := FALSE );
			FB_WriteFile_Datalog(	sNetId:='169.254.147.163.1.1',
			hFile:=FB_OpenFile_Datalog.hFile,
			pWriteBuff:= ADR(LogData),
			cbWriteLen:= LEN(LogData),		(*	i_len,	*)
			bExecute:=TRUE,
			tTimeout:=T#2s );
			nstep := nstep + 1;

	5:		FB_WriteFile_Datalog( bExecute := FALSE );
			IF ( NOT FB_WriteFile_Datalog.bBusy ) THEN
			IF ( FB_WriteFile_Datalog.bError ) THEN
			nFB_WriteFile_Datalog_ErrId := FB_WriteFile_Datalog.nErrId;
			bErrorDataLog := TRUE;
			nstep := 50;
			ELSE
			hDataLogSrcFile := FB_OpenFile_Datalog.hFile;
			nstep := nstep + 1;
			END_IF
			END_IF

	6:(* close the destination file *)
			FB_CloseFile_Datalog( bExecute := FALSE );
			FB_CloseFile_Datalog( 	sNetId:='169.254.147.163.1.1' ,
			hFile:=FB_OpenFile_Datalog.hFile,
			bExecute:=TRUE,
			tTimeout:=T#2s );
			nstep := nstep + 1;

	7:		FB_CloseFile_Datalog( bExecute := FALSE );
			IF ( NOT FB_CloseFile_Datalog.bBusy ) THEN
			IF ( FB_CloseFile_Datalog.bError ) THEN
			nFB_CloseFile_Datalog_ErrId := FB_CloseFile_Datalog.nErrId;
			bErrorDataLog := TRUE;
			END_IF
			nstep := 0;
			END_IF

END_CASE
END_FUNCTION_BLOCK

(* POU Auto/ColomnPushPiston_XY, ST *)
PROGRAM ColomnPushPiston_XY
VAR
	R_TRIG_1: R_TRIG;
	ColoumnConeCounter: CTU;
	bQAConePushPistonY: BOOL;
	step1: INT;

	step2: INT;
	PushPistonXFwdDly2: TON;
	bQAColumnPushPistonValve2: BOOL;
	bQAColumnPushPistonValve1: BOOL;
	PushPistonXFwdDly1: TON;
	temp1: BOOL;
	bAColumnPushPistonStartBit1: BOOL;
	bSetHmiSelected: BOOL;
	bAColumnPushPistonStartBit2: BOOL;
	bAColumnPushPistonStartBit1temp: BOOL;
	bAColumnPushPistonStartBit2temp: BOOL;
	bMCStart1temp: BOOL;
	bMCStart2temp: BOOL;
	bResetPushPiston: BOOL;
	StopStep: INT;
	ColumnPushCylFwdRsErrChk: RS_Error;
	ColumnPushCylFwdRsErr: BOOL;
	test: BOOL;
END_VAR
bQAColumnPushPistonValveY:=(bQAColumnPushPistonValveY1 OR bQAColumnPushPistonValveY2);

bQAColumnPushPistonValve:= ( bQAColumnPushPistonValve1 OR bQAColumnPushPistonValve2);

bAColumnPushPistonStartBit1:= ( bAColumnPushPistonStart1 OR bAColumnPushPistonStart1_23);

bAColumnPushPistonStartBit2:=( bAColumnPushPistonStart2 OR bAColumnPushPistonStart2_23);

bSetHmiSelected:=( b2_4SetHmiSelected OR b2_3SetHmiSelected );


CASE step1 OF

	0:	IF  bAutoModeOn THEN
		bQAColumnPushPistonValveY1:=TRUE;
		bColumnPushPistonReset:=FALSE;
		PushPistonXFwdDly1(IN:=FALSE); step1:=step1+1;
		ELSE
		bQAColumnPushPistonValveY1:=FALSE;
		END_IF  sMessage_Colomn:='     ';

	1:(*	IF  bAutoModeOn AND bSetHmiSelected AND NOT bAPauseSeq AND bAColumnPushPistonStartBit1 AND bIColumnPushPistonHome  AND NOT bQASealingConveyorMotor  AND NOT bIRowConeCountSensor AND NOT bQAMatrixConveyorMotor  AND ( bMCStart1 OR bMCStart2 ) THEN
		PushPistonXFwdDly1(IN:=FALSE); *)
		bQAColumnPushPistonValveY1:=TRUE; step1:=step1+1;  sMessage_Colomn:='     ';
		(*END_IF*)

	2:	IF  bAutoModeOn AND bSetHmiSelected AND NOT bAPauseSeq AND bAColumnPushPistonStartBit1 AND bIColumnPushPistonHome
		AND NOT bQASealingConveyorMotor  AND NOT bIRowConeCountSensor AND NOT bQAMatrixConveyorMotor AND NOT bAConeMissAtMatricConv AND
		 NOT bIRowConeDetection  AND ( bMCStart1 OR bMCStart2 OR bWCSStart1_24 OR bWCSStart2_24 )  AND NOT bOneSetReached   THEN
		bQAColumnPushPistonValveY1:=FALSE;
		bColumnPushPistonReset:=FALSE;step1:=step1+1;
		END_IF   sMessage_Colomn:='Check ColumnPush Piston Home  Reed Switch';

	3:	PushPistonXFwdDly1(IN:=TRUE , PT:=t#1s , Q=> , ET=> );
		IF  PushPistonXFwdDly1.Q THEN
		bMCStart1:=FALSE;
		bMCStart2:=FALSE;step1:=step1+1;
		END_IF  sMessage_Colomn:='     ';

	4:	IF NOT bAPauseSeq  THEN step1:=step1+1; END_IF

	5:	bQAColumnPushPistonValve1:=TRUE;
		bAColumnPushPistonStart1:=FALSE;
		bAColumnPushPistonStart1_23:=FALSE;
		step1:=step1+1;

	6:	step1:=step1+1;

	7:	IF bIColumnPushPistonEnd AND NOT bAPauseSeq AND NOT bAColumnPushPistnRsError  AND NOT bAConeMissAtMatricConv THEN
		bQAColumnPushPistonValve1:=FALSE;
		bAMatrixConvStart1:=TRUE;step1:=step1+1;
		END_IF

	8:	 step1:=step1+1;

	9:	IF bIColumnPushPistonHome  AND NOT bAPauseSeq  THEN
		bQAColumnPushPistonValveY1:=TRUE;step1:=step1+1;
		END_IF  sMessage_Colomn:='Check ColumnPush Piston Home  Reed Switch';

	10:	step1:=step1+1;

	11:	PushPistonXFwdDly1(IN:=FALSE);
		bAFirstSetToMatrix:=TRUE;
		step1:=step1+1;  sMessage_Colomn:='     ';

	12:	step1:=0;  sMessage_Colomn:='     ';

END_CASE



CASE step2 OF



	0:	IF  bAutoModeOn AND bSetHmiSelected AND bAColumnPushPistonStartBit2  AND bIColumnPushPistonHome
		AND NOT bQASealingConveyorMotor  AND bAFirst3ConeAtRowConeCountTemp  AND NOT bAConeMissAtMatricConv  THEN
		PushPistonXFwdDly2(IN:=FALSE);
		bQAColumnPushPistonValveY1:=FALSE;step2:=step2+1;
		END_IF   sMessage_Colomn:='Check ColumnPush Piston Home  Reed Switch';

	1:	IF NOT bAPauseSeq THEN step2:=step2+1; END_IF

	2:	PushPistonXFwdDly2(IN:=TRUE , PT:=t#1s , Q=> , ET=> );   (* PT:=t#0.3s *)
		IF  PushPistonXFwdDly2.Q THEN
		step2:=step2+1;
		END_IF

	3:	IF NOT bAPauseSeq THEN step2:=step2+1; END_IF

	4:	bQAColumnPushPistonValve2:=TRUE;
		bAColumnPushPistonStart2:=FALSE;
		bAColumnPushPistonStart2_23:=FALSE;
		step2:=step2+1;

	5:	IF NOT bAPauseSeq THEN step2:=step2+1; END_IF

	6:	IF bIColumnPushPistonEnd AND NOT bAColumnPushPistnRsError THEN
		bQAColumnPushPistonValve2:=FALSE;
		bAMatrixConvStart2:=TRUE;
		step2:=step2+1;
		END_IF


	7:	IF NOT bAPauseSeq THEN step2:=step2+1; END_IF

	8:	IF bIColumnPushPistonHome  THEN
		bQAColumnPushPistonValveY1:=TRUE;
		step2:=step2+1;
		END_IF   sMessage_Colomn:='Check ColumnPush Piston Home  Reed Switch';

	9:	IF NOT bAPauseSeq THEN step2:=step2+1; END_IF

	10:	PushPistonXFwdDly2(IN:=FALSE);
		bASecondSetToMatrix:=TRUE;
		step2:=step2+1;

	11:	IF NOT bAPauseSeq THEN step2:=step2+1; END_IF

	12:	step2:=0;

END_CASE

CASE StopStep OF

0:	IF NOT  bIEmergencySwitch OR  bStopHmi  OR bServoOff OR bIMcStop   THEN
	step1:=0;
	step2:=0;
	bAColumnPushPistonStart1:=FALSE;
	bAColumnPushPistonStart1_23:=FALSE;
	bAColumnPushPistonStart2:=FALSE;
	bAColumnPushPistonStart2_23:=FALSE;
	bAColumnPushPistonStartBit1:=FALSE;
	bAColumnPushPistonStartBit2:=FALSE;
	bQAColumnPushPistonValve1:=FALSE;
	bQAColumnPushPistonValve2:=FALSE;
	bResetPushPiston:=TRUE;
	bAMatrixConvStart1:=FALSE;
	bAMatrixConvStart2:=FALSE;
	StopStep:=1;
         CoinCheckBeforMatrix:=FALSE;

	END_IF

1:	IF bResetPushPiston AND bIColumnPushPistonHome THEN
	bQAColumnPushPistonValveY1:=FALSE;
	bQAColumnPushPistonValveY2:=FALSE;
	bColumnPushPistonReset:=TRUE;
	bResetPushPiston:=FALSE;
	StopStep:=0;
	END_IF
END_CASE




IF  bAutoModeOn AND bSetHmiSelected  AND bAColumnPushPistonStartBit1 AND bIColumnPushPistonHome
		AND NOT bQASealingConveyorMotor  AND NOT bIRowConeCountSensor AND NOT bQAMatrixConveyorMotor AND NOT bAConeMissAtMatricConv
		 AND  bIRowConeDetection  AND ( bMCStart1 OR bMCStart2 OR bWCSStart1_24 OR bWCSStart2_24 ) THEN
		CoinCheckBeforMatrix:=TRUE; sMatrixConvStatus:='Clear Cone At Matrix Conveyor'; END_IF

IF CoinCheckBeforMatrix AND bAutoModeOn AND bErrorReset  AND NOT bIRowConeDetection  THEN
 sMatrixConvStatus:=''; CoinCheckBeforMatrix:=FALSE;END_IF
END_PROGRAM

(* POU Auto/Matrix_Conveyor, ST *)
PROGRAM Matrix_Conveyor
VAR
	step1: INT;
	tMatrixConvStopDly: TON;

	step2: INT;
	bMatrixConvlUnitIntOverTemp: BOOL;
	bIColumnPushPistonEndtemp: BOOL;
	test: BOOL;
	bAConeAtMatrixCon: BOOL;
END_VAR
bQAMatrixConveyorMotor:=( bQAMatrixConveyor1 OR bQAMatrixConveyor2 );

CASE step1 OF

	0:	IF bIColumnPushPistonEnd AND bAutoModeOn  AND bAMatrixConvStart1 AND NOT bAPauseSeq  AND NOT bAColumnPushPistnRsError   THEN
		step1:=step1+1;
		END_IF

	1:	IF  NOT  bAConeOnMatrixConv AND NOT bIRowConeDetection AND NOT bOneSetReached  THEN  bQAMatrixConveyor1:=TRUE; step1:=step1+1 ; END_IF

	2:	IF bIRowConeCountSensor THEN
		bQAMatrixConveyor1:=FALSE;
		bAMatrixConvStart1:=FALSE;
		tMatrixConvStopDly(IN:=FALSE);
		step1:=step1+1;
		END_IF

	3:	IF NOT bIRowConeDetection AND NOT bAConeOnMatrixConv OR NOT bAConeAtMatrixCon OR NOT  bConeAtMatrixConveter THEN
 		bAFirst3ConeAtRowConeCount:=TRUE;
		bAFirst3ConeAtRowConeCountTemp:=TRUE;
		step1:=step1+1; END_IF

	4:	IF bIColumnPushPistonEnd THEN step1:=step1+1; END_IF

	5:	IF bAutoModeOn AND  bAMatrixConvStart2   AND( bRowStopperAt23Pos OR bRowStopperAt24Pos) AND NOT bAPauseSeq
		 AND NOT bAColumnPushPistnRsError AND NOT bAConeAtMatrixCon AND NOT bIRowConeDetection THEN
		bQAMatrixConveyor2:=TRUE;
		bAFirst3ConeAtRowConeCountTemp:=FALSE;
		step1:=step1+1;
		END_IF

	6:	bAMatrixConvStart2:=FALSE;
		bRowStopperAt23Pos:=FALSE;
		bRowStopperAt24Pos:=FALSE;
		 step1:=step1+1;

	7: 	IF bIRowConeDetection AND bAutoModeOn THEN
		tMatrixConvStopDly(IN:=TRUE , PT:=t#0.7s , Q=> , ET=> );
		IF tMatrixConvStopDly.Q THEN  step1:=step1+1; END_IF
		END_IF

	8:	 step1:=step1+1;

	9:	bARowStopperMotorRevStart:=TRUE;
		bQAMatrixConveyor2:=FALSE;
		bOneSetReached:=TRUE;
		step1:=0;
END_CASE


(*==========First Cone Missed========*)

IF bAFirst3ConeAtRowConeCount  AND( bIRowConeCountSensor AND bIRowConeDetection)THEN
bAConeAtMatrixCon:=TRUE;
 sMatrixConvStatus:='Clear Cone At Matrix Conveyor';
 bAFirst3ConeAtRowConeCount:=FALSE; END_IF

IF bAConeAtMatrixCon AND bAutoModeOn AND bErrorReset  AND NOT bIRowConeDetection  THEN
 sMatrixConvStatus:=''; bAConeAtMatrixCon:=FALSE;END_IF

IF bAConeOnMatrixConv OR bAConeAtMatrixCon OR bConeAtMatrixConveter OR CoinCheckBeforMatrix THEN
 bAConeMissAtMatricConv:=TRUE; ELSE bAConeMissAtMatricConv:=FALSE; END_IF




IF bRowStopperIntOver THEN
bMatrixConvlUnitIntOverTemp:=TRUE;
END_IF






CASE step2 OF


	0:	IF bMatrixConvlUnitIntOverTemp THEN Step2:=Step2+1; END_IF

	1:	bMCStart1:=TRUE; Step2:=Step2+1;

	2:	IF  bAFirstSetToMatrix THEN
		bMatrixConvlUnitIntOverTemp:=FALSE ; Step2:=Step2+1;END_IF

	3:	IF bOneSetReached AND ( bRowStopperAt23Pos OR bRowStopperAt24Pos ) THEN
		bMCStart2:=TRUE;Step2:=Step2+1;END_IF

	4:	bOneSetReached:=FALSE;Step2:=Step2+1;

	5:	Step2:=2;

END_CASE


IF NOT bIEmergencySwitch OR bStopHmi   OR bServoOff OR bIMcStop   THEN
bAMatrixConvStart2:=FALSE;
bRowStopperAt23Pos:=FALSE;
bRowStopperAt24Pos:=FALSE;
bMatrixConvlUnitIntOverTemp:=FALSE;
bQAMatrixConveyor1:=FALSE;
bQAMatrixConveyor2:=FALSE;
bOneSetReached:=FALSE;
bRowStopperIntOver:=FALSE;
bAFirst3ConeAtRowConeCount:=FALSE;
bAFirst3ConeAtRowConeCountTemp:=FALSE;
bQAMatrixConveyor2:=FALSE;
tMatrixConvStopDly(IN:=FALSE);
bARowStopperMotorRevStart:=FALSE;
bAConeMissAtMatricConv:=FALSE;
bOneSetReached:=FALSE;
bAConeAtMatrixCon:=FALSE;
sMatrixConvStatus:='Continue Machine Operation';
bAFirstSetToMatrix:=FALSE;
bAConeOnMatrixConv:=FALSE;
bMCStart2:=FALSE;
bMCStart1:=FALSE;
step1:=0;
Step2:=0;
bAMatrixConvStart1:=FALSE;
END_IF
END_PROGRAM

(* POU Auto/CartonConveyor, ST *)
PROGRAM CartonConveyor
VAR
	step: INT;
	bQACartonFeedingPistonValveOn1: BOOL;

	bQACartonConveyorMotor1: BOOL;
	bQACartonConveyorMotor2: BOOL;
	F_TRIG_1: F_TRIG;
	bACartonConvOffAuto: BOOL;
	bICartonFeedingPistonEndTemp: BOOL;
	TEST: BOOL;
	Timer1: TON;
	CartonTimer: TON;
	CartonStopTimer: TON;
	CartonTimer_1: TON;
	CartonTimer_2: TON;
	Carton2Timer: TON;
END_VAR
IF NOT bIEmergencySwitch OR   bStopHmi OR bServoOff  OR bIMcStop  THEN
bQACartonConveyorMotor:=FALSE;
step:=0;
bQACartonConveyorMotor1:=FALSE;
bACartonReady_23:=FALSE;
bACartonReady_24:=FALSE;
bQACartonConveyorMotor2:=FALSE;
bAEmptyCartonConvContinue:=FALSE;
bAGripperSeqover:=FALSE;
bAOneMinConvStart:=FALSE;
bACartonConvOffAuto:=FALSE;
 bHmiColourChangeBit2_24:=FALSE;
CartonTimer(IN:=FALSE);
END_IF


IF bAInitializeSeq THEN
step:=0;

END_IF




(*
bQACartonFeedingPistonValve:= (bQACartonFeedingPistonValveOn1 );
s

*)
bQACartonConveyorMotor:= (bQACartonConveyorMotor1 OR bQACartonConveyorMotor2  );



CASE step OF


	0: 	IF bAutoModeOn AND bICartonFeedingPistonHome AND bAStartCartonCov (* AND NOT bQEmptyCartonConveyorMotor *)AND NOT bAPauseSeq THEN
		bQACartonConveyorMotor1:=TRUE;
		CartonStopTimer(IN:=FALSE);
		step:=step+1;
		END_IF sMessage_Carton:='  Check Carton Feeding Home Reed Switch ';

	1:	IF bAutoModeOn AND b2_3SetHmiSelected THEN
		step:=step+1;
		sMessage_Carton:='        ';
		ELSIF  bAutoModeOn AND b2_4SetHmiSelected THEN
		step:=step+4;
		END_IF  sMessage_Carton:='       ';

	2:	IF bAutoModeOn AND  b2_3SetHmiSelected AND b2_3_BCartonHMI THEN  step:=step+1;
		ELSIF  bAutoModeOn AND  b2_3SetHmiSelected AND b2_3_ACartonHMI THEN  step:=step+2; END_IF


	3:	IF bAutoModeOn AND  b2_3SetHmiSelected AND   bICartonPosition1 THEN
		bAStartCartonCov:=FALSE;
		bQACartonConveyorMotor1:=FALSE;
		bACartonReady_23:=TRUE;
		step:=step+3;
		END_IF

	4:	IF  bAutoModeOn AND  b2_3SetHmiSelected AND  bICartonPosition3 THEN
		CartonStopTimer(IN:=TRUE  , PT:=t#0.5s , Q=> , ET=> );
		IF CartonStopTimer.Q THEN
		bAStartCartonCov:=FALSE;
		bQACartonConveyorMotor1:=FALSE;
		bACartonReady_23:=TRUE;
		step:=step+2;
		END_IF END_IF

	5:	IF bAutoModeOn AND  b2_4SetHmiSelected AND bICartonPosition2 THEN
		bQACartonConveyorMotor1:=FALSE;
		bACartonReady_24:=TRUE;
		bAStartCartonCov:=FALSE;
		step:=step+1;
		END_IF

	6:	 IF  bAGripperSeqover AND bAOneMinConvReady AND bAutoModeOn  AND NOT bAPauseSeq    THEN
		bQACartonConveyorMotor2:=TRUE;
		CartonStopTimer(IN:=FALSE);
		Carton2Timer(IN:=FALSE);
		step:=step+1;
		END_IF


	7:	IF bIFullCartonCountingSensor THEN bAOneMinConvStart:=TRUE; bAOneMinConvReady:=FALSE; step:=step+1; END_IF    (*=============== Newly Added on 04.10.16======*)

	8:	IF  bIFullCartonCountingSensor AND NOT bICartonPosition1 AND NOT bICartonPosition2 AND NOT bICartonPosition3  THEN step:=step+1; END_IF

	9: 	IF NOT bIFullCartonCountingSensor  AND  NOT bICartonPosition1 AND NOT bICartonPosition2 AND NOT bICartonPosition3 THEN step:=step+1; END_IF     (*=============== Newly Added on 04.10.16======*)

	10:	IF bACartonConvOffAuto AND bAutoModeOn   AND NOT bAPauseSeq THEN            (*===== old Pgm   bQACartonConveyorMotor2:=FALSE;*)

		bAEmptyCartonConvContinue:=TRUE;
		bAGripperSeqover:=FALSE;

		step:=step+1;
		END_IF

	11:	IF bAutoModeOn AND  b2_3SetHmiSelected AND  b2_3_BCartonHMI AND  bICartonPosition1  THEN   (*======OLD Pgm bACartonConvOffAuto:=FALSE; step:=0;*)
		bACartonConvOffAuto:=FALSE;
		CartonStopTimer(IN:=FALSE);
		bQACartonConveyorMotor2:=FALSE;
		bACartonReady_23:=TRUE;
		step:=6; sMessage_Carton:='       ';
		ELSIF bAutoModeOn AND  b2_3SetHmiSelected AND b2_3_ACartonHMI  AND bICartonPosition3 THEN   (*======OLD Pgm bACartonConvOffAuto:=FALSE; step:=0;*)
		bACartonConvOffAuto:=FALSE;
		CartonStopTimer(IN:=FALSE);
		bQACartonConveyorMotor2:=FALSE;
		bACartonReady_23:=TRUE;
		step:=11; sMessage_Carton:='       ';
		ELSIF bAutoModeOn AND   b2_4SetHmiSelected AND bICartonPosition2  THEN   (*======OLD Pgm bACartonConvOffAuto:=FALSE; step:=0;*)
		bACartonConvOffAuto:=FALSE;
		CartonStopTimer(IN:=FALSE);
		bQACartonConveyorMotor2:=FALSE;
		bACartonReady_24:=TRUE;
		step:=6; sMessage_Carton:='       ';
		END_IF sMessage_Carton:='       ';

	12:  Carton2Timer(IN:=TRUE  , PT:=t#0.5s , Q=> , ET=> );
		IF Carton2Timer.Q THEN step:=6; END_IF

END_CASE

IF bACartonReady_24 AND b2_4SetHmiSelected AND NOT bICartonPosition2 AND NOT bQACartonConveyorMotor2 AND NOT bQACartonConveyorMotor1  THEN
CartonTimer(IN:=TRUE  , PT:=t#0.4s , Q=> , ET=> ); ELSE CartonTimer(IN:=FALSE);
END_IF

IF bACartonReady_23 AND b2_3SetHmiSelected AND NOT bICartonPosition1 AND b2_3_BCartonHMI AND NOT bQACartonConveyorMotor2 AND NOT bQACartonConveyorMotor1 THEN
CartonTimer_1(IN:=TRUE  , PT:=t#0.4s , Q=> , ET=> ); ELSE CartonTimer_1(IN:=FALSE);
END_IF

IF bACartonReady_23 AND b2_3SetHmiSelected AND NOT bICartonPosition3 AND b2_3_ACartonHMI  AND NOT bQACartonConveyorMotor2 AND NOT bQACartonConveyorMotor1 THEN
CartonTimer_2(IN:=TRUE  , PT:=t#0.4s , Q=> , ET=> ); ELSE CartonTimer_2(IN:=FALSE);
END_IF




IF( CartonTimer.Q OR CartonTimer_1.Q OR CartonTimer_2.Q)  THEN  HmiFullCartonAtConveyer_sensor:='Aline the  Carton  At Full Carton Conveyor';
 bHmiColourChangeBit2_24:=TRUE;
ELSIF (bICartonPosition2 OR bICartonPosition1 )  AND (bErrorReset  )THEN
 CartonTimer(IN:=FALSE); HmiFullCartonAtConveyer_sensor:=' Continue Machine Operation';
CartonTimer_1(IN:=FALSE);
CartonTimer_2(IN:=FALSE);
 bHmiColourChangeBit2_24:=FALSE;

END_IF

(*
		IF bISeparatorVerticalPistonHome AND bAutoModeOn THEN
		bAGripperSeqover:=TRUE;
		END_IF

*)

F_TRIG_1(CLK:=bIFullCartonCountingSensor , Q=> );

		IF F_TRIG_1.Q AND bQACartonConveyorMotor2 THEN
		bACartonConvOffAuto:=TRUE;
		END_IF


IF  b2_3SetHmiSelected  AND b2_3_BCarton  THEN 	b2_3_ACartonHMI:=FALSE; b2_3_BCartonHMI:=TRUE;  END_IF

IF  b2_3SetHmiSelected AND b2_3_ACarton THEN 	b2_3_ACartonHMI:=TRUE; b2_3_BCartonHMI:=FALSE; END_IF

IF  b2_4SetHmiSelected  THEN 	b2_3_ACartonHMI:=FALSE; b2_3_BCartonHMI:=FALSE; END_IF
END_PROGRAM

(* POU Auto/EmptyConveyor, ST *)
PROGRAM EmptyConveyor
VAR
	start: BOOL;
	bQACartonFeedingPistonValve1: BOOL;
	bQACartonFeedingPistonValve2: BOOL;
	Step: INT;
	bLocalReset: BOOL;
	startEmptyConv: BOOL;

END_VAR
IF bAInitializeSeq THEN

step:=0;

END_IF
bQAEmptyCartonConveyorMotor:= (bQAEmptyCartonConveyorMotor1 );


bQACartonFeedingPistonValve:= ( bQACartonFeedingPistonValve1 OR bQACartonFeedingPistonValve2 );
(*==========Empty Conveyor First Start==================*)




		IF ( (*bMCStartInAuto OR  *)  bClearConeInt )AND  ( b2_3SetHmiSelected OR b2_4SetHmiSelected )  AND bIGripperVerticalHome AND NOT bAPauseSeq
		   THEN startEmptyConv:=TRUE; 	  END_IF

		IF bManualModeOn OR bIMcStop   THEN startEmptyConv:=FALSE;  END_IF (*not changed*)

		IF bAutoModeOn AND startEmptyConv AND NOT bIEmptyCartonDetectionSensor  AND NOT bQACartonFeedingPistonValve AND bICartonFeedingPistonHome THEN
		bQAEmptyCartonConveyorMotor1:=TRUE;
		bAIntStarted:=FALSE;
		ELSE
		bQAEmptyCartonConveyorMotor1:=FALSE;
		END_IF

CASE Step OF


	0:  IF b2_4SetHmiSelected  THEN
		step:=step+1;
		ELSIF b2_3SetHmiSelected THEN
		step:=step+1;
		END_IF

	1:	IF NOT bAPauseSeq THEN step:=step+1; END_IF

	2:	IF bAutoModeOn AND startEmptyConv AND  bIEmptyCartonDetectionSensor  AND NOT bQACartonConveyorMotor AND NOT bICartonPosition1
		  AND NOT bICartonPosition2  AND NOT bICartonPosition3  AND NOT bIFullCartonCountingSensor AND NOT bCartonFullDetectbit
		AND NOT bEmptyCartonDetectError THEN
		bQACartonFeedingPistonValve1:=TRUE;
		bClearConeInt:=FALSE;
		step:=step+1;
		END_IF

	3:	IF NOT bAPauseSeq THEN step:=step+1; END_IF

	4:	IF bAutoModeOn AND startEmptyConv AND NOT bIEmptyCartonDetectionSensor  AND  bICartonFeedingPistonEnd  THEN
		bQACartonFeedingPistonValve1:=FALSE;
		bAStartCartonCov:=TRUE;
		step:=step+1;
		END_IF

	5:	IF NOT bAPauseSeq THEN step:=step+1; END_IF

	6:	IF bAutoModeOn AND bAEmptyCartonConvContinue AND  bIEmptyCartonDetectionSensor (*AND NOT bQACartonConveyorMotor *)
		AND NOT bICartonPosition1  AND NOT bICartonPosition2 AND NOT bICartonPosition3  AND NOT bIFullCartonCountingSensor
		AND NOT bEmptyCartonDetectError  THEN
		bQACartonFeedingPistonValve2:=TRUE;     (*===== it was included===AND NOT bQACartonConveyorMotor*)
		step:=step+1;
		END_IF

	7:	IF NOT bAPauseSeq THEN step:=step+1; END_IF

	8:	IF bAutoModeOn AND startEmptyConv AND NOT bIEmptyCartonDetectionSensor  AND  bICartonFeedingPistonEnd  THEN
		bQACartonFeedingPistonValve2:=FALSE;
		bAStartCartonCov:=TRUE;
		step:=step+1;
		END_IF

	9:	IF NOT bAPauseSeq THEN step:=step+1; END_IF

	10:	bAEmptyCartonConvContinue:=FALSE;
		step:=6;

END_CASE


IF NOT bIEmergencySwitch OR bStopHmi   OR bServoOff  OR bIMcStop  THEN
step:=0;
bQAEmptyCartonConveyorMotor1:=FALSE;
bQACartonFeedingPistonValve1:=FALSE;
bQACartonFeedingPistonValve2:=FALSE;
bAEmptyCartonConvContinue:=FALSE;
bAStartCartonCov:=FALSE;
startEmptyConv:=FALSE;
bClearConeInt:=FALSE;
bEmptyCartonDetectError:=FALSE;
		bAIntStarted:=FALSE;
END_IF
END_PROGRAM

(* POU Auto1/SeparatorUnit, ST *)
PROGRAM SeparatorUnit
VAR
	n1: INT;
	n2: INT;
	n3: INT;
	bASeparator1Enable: BOOL;
	Count: INT;
	bASeparator2Enable: BOOL;
	bASeparator3Enable: BOOL;
	bASeparatorEnabled: BOOL;
	step: INT;
	bQASeparatorVerticalPistonOnAuto: BOOL;
	TON_1: TON;
	bQAVacuumPistonValveOnAuto: BOOL;
	TON_2: TON;
	TON_3: TON;
	bASeparatorUnitEnableTemp: BOOL;
	bASeparatorEnabledTemp: BOOL;
	bISeparatorVerticalPistonHomeTemp: BOOL;
	bISeparatorVerticalPistonEndTemp: BOOL;
	OpCount: INT;
	VerSepCylHomeRsErrChk: RS_Error;
	VerSepCylHomeRsErr: BOOL;
	SepPickSenErrChk: RS_Error;
	OpCountTemp: INT;
	SelectLayer_1: SelectLayer;
	iTotalLayersTemp: INT;
	bAGripperSeqover1: BOOL;
	bAGripperSeqover2: BOOL;
	bAGripperSeqover1temp: BOOL;
	OpCountRst: TON;
END_VAR
bQASeparatorVerticalPistonValve:= ( bQASeparatorVerticalPistonOnAuto );

bQAVacuumPistonValve:= ( bQAVacuumPistonValveOnAuto );



CASE step OF


	0:	TON_1(IN:= FALSE);
		 step:=step+1;


	1:	step:=step+1;

	2:	IF bAutoModeOn AND bASeparatorUnitEnable AND bISeparatorHorizontalPistonHome AND bASeparatorEnabled
		 AND bISeparatorVerticalPistonHome AND NOT bAPauseSeq   THEN
		TON_1(IN:= TRUE , PT:=T#0.5S , Q=> , ET=> );
		IF TON_1.Q THEN step:=step+1; END_IF
		END_IF   sMessage_Separator:='   Check Separator Horizontal & Vertical  Piston Home Reed Switch    ';


	3:	 step:=step+1;

	4:	bQASeparatorVerticalPistonOnAuto:=TRUE;
		bASeparatorUnitEnable1:=FALSE;
		bASeparatorUnitEnable2:=FALSE;
		bASeparatorUnitEnable3:=FALSE;
		bASeparatorUnitEnable:=FALSE;
		TON_1(IN:= FALSE);
		TON_2(IN:=FALSE);
		step:=Step+1; sMessage_Separator:='            ';

	5:	IF bISeparatorPickupDetectionSensor  THEN step:=step+1; END_IF

	6:	IF NOT bAPauseSeq THEN
		bQAVacuumPistonValveOnAuto:=TRUE;
		step:=Step+1;
		END_IF sMessage_Separator:='            ';

	7:	step:=step+1;

	8:	TON_2(IN:=TRUE , PT:=T#0.1s , Q=> , ET=> );
		IF TON_2.Q THEN step:=step+1; END_IF

	9:	IF NOT bAPauseSeq THEN step:=step+1; END_IF

	10:	bQASeparatorVerticalPistonOnAuto:=FALSE;
		bASepVerticalCylRevRsErrChkBit:=TRUE;
		step:=Step+1;

	11:	 step:=step+1;

	12:	IF bAutoModeOn AND	bISeparatorHorizontalPistonEnd   (*AND bASeparatorEnabled  *) AND bISeparatorVerticalPistonHome
		 AND NOT  bAPauseSeq AND NOT bASepaVerCylhomeRsError THEN
		bQASeparatorVerticalPistonOnAuto:=TRUE;
		bASepVerticalCylRevRsErrChkBit:=FALSE;
		bASepVerticalCylEndRsErrChkBit:=TRUE;
		TON_2(IN:=FALSE);
		TON_3(IN:= FALSE);
		step:=step+1;
		END_IF  sMessage_Separator:='   Check Separator  Vertical  Piston Home Reed Switch    ';

	13:	   step:=step+1;

	14:	IF bISeparatorVerticalPistonEnd THEN

		step:=step+1;
		END_IF

	15: IF NOT bASepaVertiEndPistnRsError  THEN  step:=step+1; END_IF sMessage_Separator:='            ';

	16:	(*IF NOT bAPauseSeq THEN*) bQAVacuumPistonValveOnAuto:=FALSE; bASepVerticalCylEndRsErrChkBit:=FALSE;
		 bSeparatorVerticalPistonEndRsSensed:=FALSE;
		step:=step+1;
		(*END_IF*)

	17:	step:=step+1;

	18:	TON_3(IN:= TRUE , PT:= T#0.5S, Q=> , ET=> );
		IF TON_3.Q THEN step:=step+1; END_IF


	19:	step:=step+1;

	20:	IF NOT bAPauseSeq THEN  bQASeparatorVerticalPistonOnAuto:=FALSE;
		TON_3(IN:= FALSE);
		step:=step+1;
		END_IF

	21:	 step:=step+1;

	22:	IF bISeparatorVerticalPistonHome THEN
		step:=step+1;
		END_IF   sMessage_Separator:='   Check Separator Vertical  Piston Home Reed Switch    ';

	23:	OpCount:=OpCount+1;
		step:=Step+1;

	24: (*	IF OpCount=iTotalLayersTemp AND  iACountServoToSepUnit =3    THEN
		bAGripperSeqover1:=TRUE;
		OpCount:=0;
		CountServo:=0;
		step:=Step+1;
		ELSIF OpCount<3 THEN
		END_IF*)
		step:=step+1;


	25:	bAGripperSeqover1:=FALSE;
		step:=0;  sMessage_Separator:='            ';



END_CASE



		IF OpCount=iTotalLayersTemp AND  iACountServoToSepUnit =3    THEN
		bAGripperSeqover1:=TRUE;
		END_IF


IF bAGripperSeqover1 OR bAGripperSeqover2  AND bAutoModeOn THEN
bAGripperSeqover:=TRUE; iACountServoToSepUnit:=0; bAGripperSeqover1:=FALSE;
 bAGripperSeqover2:=FALSE; bACartonReady_23:=FALSE;
bACartonReady_24:=FALSE;
END_IF

IF bAGripperSeqover THEN OpCount:=0; OpCountRst(IN:=TRUE , PT:=t#0.1s , Q=> , ET=> ); bASeparatorUnitEnable:=FALSE;bASeparatorUnitEnable2:=FALSE;
bASeparatorUnitEnable1:=FALSE;  END_IF
IF OpCountRst.Q THEN CountServo:=0; OpCountRst(IN:=FALSE); END_IF
SelectLayer_1(
	bVarIn1:=bALayer1Selected ,(*1*)
	 bVarIn2:= bALayer2Selected,(*2*)
	 bVarIn3:= bALayer3Selected, (*4*)
	ByteResult=> iTotalLayers );


IF iTotalLayers = 7 THEN iTotalLayersTemp:=3 ;
ELSIF iTotalLayers = 6 THEN iTotalLayersTemp:=2 ;
ELSIF iTotalLayers = 5 THEN iTotalLayersTemp:=2 ;
ELSIF iTotalLayers = 4 THEN iTotalLayersTemp:=1 ;
ELSIF iTotalLayers = 3 THEN iTotalLayersTemp:=2 ;
ELSIF iTotalLayers = 2 THEN iTotalLayersTemp:=1 ;
ELSIF iTotalLayers = 1 THEN iTotalLayersTemp:=1 ;
ELSIF iTotalLayers =0  THEN iTotalLayersTemp:=0 ;
END_IF

iTotalLayersHold:=iTotalLayers;

IF bAutoModeOn AND iTotalLayersTemp = 0 AND iACountServoToSepUnit = 3 THEN bAGripperSeqover2:=TRUE;  iACountServoToSepUnit:=0;    END_IF

IF bAServoDown1Done AND CountServo = 0  AND bALayer1Selected  THEN
bASeparatorUnitEnable1:=TRUE;END_IF

IF bAServoDown1Done AND CountServo = 1 AND bALayer2Selected  THEN
bASeparatorUnitEnable2:=TRUE; END_IF

IF bAServoDown1Done AND CountServo = 2  AND bALayer3Selected THEN
bASeparatorUnitEnable3:=TRUE;
END_IF

IF bASeparatorUnitEnable1 OR bASeparatorUnitEnable2 OR bASeparatorUnitEnable3 THEN bASeparatorUnitEnable:= TRUE; ELSE bASeparatorUnitEnable:=FALSE;  END_IF

(*===================  Separator Layer Enable Logic=======================*)

IF bLayer1SelectHmi THEN bALayer1Selected:=TRUE; ELSE   bALayer1Selected:=FALSE; END_IF

IF bLayer2SelectHmi THEN bALayer2Selected:=TRUE; ELSE   bALayer2Selected:=FALSE; END_IF

IF bLayer3SelectHmi THEN bALayer3Selected:=TRUE; ELSE   bALayer3Selected:=FALSE; END_IF



IF bALayer1Selected THEN n1:=1; ELSE n1:=0; END_IF

IF bALayer2Selected THEN n2:=2; ELSE n2:=0; END_IF

IF bALayer3Selected THEN n3:=3; ELSE n3:=0; END_IF




IF n1=1 AND CountServo=0 THEN bASeparator1Enable:=TRUE;  ELSE   bASeparator1Enable:=FALSE; END_IF

IF n2=2 AND CountServo=1 THEN bASeparator2Enable:=TRUE;  ELSE   bASeparator2Enable:=FALSE; END_IF

IF n3=3 AND CountServo=2 THEN bASeparator3Enable:=TRUE;  ELSE   bASeparator3Enable:=FALSE; END_IF

	IF bASeparator1Enable OR bASeparator2Enable OR bASeparator3Enable THEN
	bASeparatorEnabled:=TRUE;
	ELSE
	bASeparatorEnabled:=FALSE;
	END_IF

(*

IF NOT  bALayer1Selected AND NOT  bALayer2Selected AND NOT   bALayer3Selected  THEN iSelectedLayers:=0;

ELSIF   bALayer1Selected AND NOT bALayer2Selected AND NOT  bALayer3Selected  THEN iSelectedLayers:=1;

ELSIF NOT  bALayer1Selected AND    bALayer2Selected AND  NOT  bALayer3Selected  THEN iSelectedLayers:=2;

ELSIF NOT bALayer1Selected AND NOT  bALayer2Selected AND    bALayer3Selected THEN iSelectedLayers:=3;

ELSIF bALayer1Selected AND  bALayer2Selected AND NOT bALayer3Selected THEN iSelectedLayers:=12;

ELSIF  NOT bALayer1Selected AND  bALayer2Selected AND   bALayer3Selected  THEN iSelectedLayers:=23;

ELSIF bALayer1Selected AND NOT  bALayer2Selected AND    bALayer3Selected  THEN iSelectedLayers:=13;

ELSIF bALayer1Selected AND bALayer3Selected AND    bALayer3Selected   THEN iSelectedLayers:=123;

END_IF



*)




IF NOT bIEmergencySwitch OR bStopHmi OR  bIMcStop OR bServoOff THEN

bQASeparatorVerticalPistonOnAuto:=FALSE;
TON_1(IN:= FALSE);
TON_2(IN:=FALSE);
bQAVacuumPistonValveOnAuto:=FALSE;
bASepVerticalCylRevRsErrChkBit:=FALSE;
bASepVerticalCylEndRsErrChkBit:=FALSE;
TON_3(IN:= FALSE);
OpCount:=0;
bAGripperSeqover1:=FALSE;
CountServo:=0;
bAGripperSeqover2:=FALSE;
step:=0;

END_IF
END_PROGRAM

(* POU FunctionBlocks/SelectLayer, ST *)
FUNCTION_BLOCK SelectLayer
VAR_INPUT


	bVarIn1: BOOL;
	bVarIn2: BOOL;
	bVarIn3: BOOL;

END_VAR
VAR_OUTPUT


	ByteResult: USINT;
END_VAR
VAR

END_VAR
ByteResult.0:=bVarIn1;
ByteResult.1:=bVarIn2;
ByteResult.2:=bVarIn3;


ByteResult;
END_FUNCTION_BLOCK

(* POU Auto1/UnitA_RowStopper24, ST *)
PROGRAM UnitA_RowStopper24
VAR




	step: INT;


	CTU_1Enable: BOOL;
	R_TRIG_1: F_TRIG;
	CTU_2: CTU;
	R_TRIG_2: R_TRIG;
	tRowStopperRevDly1: TON;
	UnitAConeCrossCount: CTU;
	test: BOOL;
	bStopRetUnitA: BOOL;
	RowStopperMotorStopDly: TON;
	bRetUnitAStarttemp: BOOL;
	bAUnitAWeighOktemp: BOOL;
	RowStopperEndRSErrorDly: TON;
	bStartTemp1: BOOL;
	UnitAOverTemp: BOOL;
	RowStopperEndSenErrChk: RS_Error;
	RowStopperEndSenErr: BOOL;
	interLockStep: INT;
	UnitACompleteCheckCountCv: INT;
	bEnableBit1: BOOL;
	UnitAConeCross: CTU;
	Testtimer: TON;
	bAUnitBConeCrossingOff_2: BOOL;
	step3: INT;
	TON_7: TON;
	R_TRIG_4: R_TRIG;
	timer3: TON;

	RowStopperCountvalue: DINT;
	UnitA_3_ConeComDly: TOF;
	UnitA_2_ConeComDly: TON;
	iSensorOnVal: UINT;
	SenSelect_1: SenSelect;
	bCheckSensor: BOOL;
	iAConeCrossCount: INT;
	GetDLy: TON;
	step2: INT;
	TON_6: TON;
	step4: INT;
	TON_8: TON;
	TON_10: TON;
	bAUnitAConeCrossing_1: BOOL;
	F_TRIG_3: F_TRIG;
	TON_9: TON;
	F_TRIG_5: F_TRIG;
	tConeCrossDly: TON;
	bAUnitBConeCrossing_1_24: BOOL;
	bAUnitAConeCrossing_1_24: BOOL;
	F_TRIG_3_24: F_TRIG;
	tConeCrossDly_1_24: TON;
	CountResetBit1_24: BOOL;
END_VAR
									(*=============Checking the No. of sensors sensed================*)

IF bCheckSensor   THEN
SenSelect_1(
		bVarIn1:=bIUnitAConedetection1 ,
		bVarIn2:= bIUnitAConedetection2,
		bVarIn3:= bIUnitAConedetection3,
		ByteResult=>iSensorOnVal );

END_IF

		IF iSensorOnVal=7 THEN iAConeCrossCount:=3;
		ELSIF  iSensorOnVal=6 THEN iAConeCrossCount:=2;
		ELSIF  iSensorOnVal=5 THEN iAConeCrossCount:=2;
		ELSIF  iSensorOnVal=4 THEN iAConeCrossCount:=1;
		ELSIF  iSensorOnVal=3 THEN iAConeCrossCount:=2;
		ELSIF  iSensorOnVal=2 THEN iAConeCrossCount:=1;
		ELSIF  iSensorOnVal=1 THEN iAConeCrossCount:=1;
		END_IF


bQAUnitA_RowStopperMotorForward1:=( bQAUnitA_RowStopperMotorFwd1 OR bQAUnitA_RowStopperMotorFwd2 );

bQAUnitA_RowStopperMotorReverse1:= ( bQAUnitA_RowStopperMotorRev1 OR bRetUnitARst );

CASE step OF

	0:	IF bAutoModeOn AND bAUnitAWeighOk  AND bRetUnitAStart  AND NOT bStopEnable  AND bAinterlockinit    THEN
		UnitACompleteCheckCount.RESET:=TRUE;
		CountResetBit1_24 :=FALSE;
		step:=step+1;
		END_IF

	1:	 step:=step+1;

	2:	IF bAutoModeOn  AND UnitACompleteCheckCount.CV =0 AND NOT CountResetBit1_24 AND NOT bAPauseSeq THEN
		bAConvFirstStart:=TRUE;
		UnitACompleteCheckCount.RESET:=FALSE;
		step:=step+1;
		END_IF

	3:	 step:=step+1;

	4:	IF bAutoModeOn    AND NOT bUnitBRowStopperStarted  AND NOT bAMainIntStarted  AND NOT bStopEnable AND NOT bAPauseSeq    THEN
		bQAUnitA_RowStopperMotorFwd1:=TRUE;
		UnitAConeCrossCount.RESET:=TRUE;
		bAUnitAWeighOk:=FALSE;
		bUnitARowStopperStarted:=TRUE;
		sRetreivalAStatus:= 'Running';
		bRetUnitAStart:=FALSE;
		 step:=step+1;
		END_IF

	5:	RowStopperMotorStopDly(In:=FALSE);
		 step:=step+1;

	6:	IF bIUnitAConedetection1 OR  bIUnitAConedetection2 OR bIUnitAConedetection3   THEN
		step:=step+1;
		ELSIF NOT bIUnitAConedetection1 AND NOT  bIUnitAConedetection2 AND NOT  bIUnitAConedetection3 AND bIUnitA_RowStopperEnd
		 THEN
		step:=14;
		END_IF

	7:	RowStopperMotorStopDly( IN:=TRUE , PT:=T#0.5s , Q=> , ET=> );IF RowStopperMotorStopDly.Q   THEN   step:=step+1; END_IF


	8:	UnitAConeCrossCount.RESET:=FALSE;
		bQAUnitA_RowStopperMotorFwd1:=FALSE;
		tRowStopperRevDly1(IN:=FALSE);
		UnitA_18_ConeComDly(IN:=FALSE);
		GetDLy(IN:=FALSE);
		step:=step+1;

	9:	IF NOT bAPauseSeq THEN  bCheckSensor:=TRUE; step:=step+1; END_IF


	10:	GetDLy(IN:=TRUE , PT:=t#0.6s , Q=> , ET=> );
		 IF GetDLy.Q THEN bCheckSensor:=FALSE;   step:=step+1;
		END_IF


	11:	IF (UnitAConeCrossCount.CV= iAConeCrossCount ) AND NOT  bIUnitA_RowStopperEnd   THEN
		RowStopperMotorStopDly(In:=FALSE);
		step:=4;
		ELSIF (* ( UnitACompleteCheckCount.CV >=  iATotalNoOfCones)*) bIUnitA_RowStopperEnd THEN
		(*UnitA_18_ConeComDly(IN:=TRUE , PT:=t#0.3s , Q=> , ET=> );
		IF UnitA_18_ConeComDly.Q THEN *) step:=step+1; 
		END_IF

	12:	IF NOT bAPauseSeq THEN step:=step+1; END_IF

	13:	IF bAutoModeOn      THEN
		bQAUnitA_RowStopperMotorFwd2:=TRUE;
		UnitA_18_ConeComDly(IN:=FALSE);
		RowStopperEndRSErrorDly(IN:=TRUE , PT:=t#5s , Q=> , ET=> );
		step:=step+1;
		END_IF

	14:	step:=step+1;

